//永久解锁动态码
IF(receive_data101[1]=16#21)THEN
	swGpsPrivate.caculateCodeH(code1:=CANO_engine_hour_h,code2:=TO_DINT(CANO_engine_hour_m),result =>CANO_DONGTAIMA1);
	swGpsPrivate.caculateCodeL(code1:=x1,code2:=x2,result =>CANO_DONGTAIMA2);
	send_data102[0]:=receive_data101[0];
	send_data102[1]:=16#21;
	send_data102[2]:=DINT_TO_BYTE((CANO_DONGTAIMA1 MOD 65536) MOD 256);
	send_data102[3]:=DINT_TO_BYTE((CANO_DONGTAIMA1 MOD 65536)/256);
	send_data102[4]:=DINT_TO_BYTE((CANO_DONGTAIMA1 / 65536) MOD 256);
	send_data102[5]:=DINT_TO_BYTE((CANO_DONGTAIMA2 MOD 65536) MOD 256);
	send_data102[6]:=DINT_TO_BYTE((CANO_DONGTAIMA2 MOD 65536)/256);
	send_data102[7]:=DINT_TO_BYTE((CANO_DONGTAIMA2 / 65536) MOD 256);
	IF tCounter<500 THEN
		tCounter:=tCounter+1;
		CAN1_SEND_102(xEnable:= TRUE, eChannel:= 0, udiID:= 16#102, xExtended:=FALSE, usiDLC:=8 , aData:=send_data102);
	ELSE
		receive_data101[1]:=0;
	END_IF
END_IF
IF(receive_data101[1]=0)THEN
	tCounter:=0;
END_IF
swGpsPrivate.swGpsPermanentCancel(PH:=CANO_DONGTAIMA1,PL:=CANO_DONGTAIMA2,result=>VarGpsYongJiuUnlockPassword2);

END_PROGRAM

// StandardPLC/Application/CAN/CAN1
PROGRAM CAN1
VAR
	CAN2_INTI: ifmRCAN.CAN_Enable;
	CANO_FUEL1 :UINT;
	CANO_FUEL2 :UINT;
	Idling_OK_biaozhi:BOOL;
	TIME_20ms:TON;
	TIME_30ms:ton;
	TIME_500ms:ton;
	TIME_5000ms:TON;
	TIME_3000ms:TON;
	TIME_1000ms:TON;
	TIME_BUTTON1:TON;
	TIME_BUTTON2:TON;
	TIME_BIAOZHI1:TON;
	TIME_GPSCAN_ERROR:TON;
	CAN2_RECE_1:ifmRCAN.CAN_Rx;
	CAN2_RECE_2:ifmRCAN.CAN_Rx;
	CAN2_RECE_3:ifmRCAN.CAN_Rx;
	CAN2_RECE_4:ifmRCAN.CAN_Rx;
	CAN2_RECE_5:ifmRCAN.CAN_Rx;
	CAN2_RECE_6:ifmRCAN.CAN_Rx;
	CAN2_RECE_7:ifmRCAN.CAN_Rx;
	CAN2_RECE_8:ifmRCAN.CAN_Rx;
	CAN2_RECE_9:ifmRCAN.CAN_Rx;
	CAN2_rece_data18FD7C00:ifmRCAN.CAN_Rx;
	CAN2_rece_data18FEFF00:ifmRCAN.CAN_Rx;
	CAN2_rece_data18FE5600:ifmRCAN.CAN_Rx;
	CAN2_SEND_000:ifmRCAN.CAN_Tx;
	CAN2_SEND_300:ifmRCAN.CAN_Tx;
	CAN2_SEND_1:ifmRCAN.CAN_Tx;
	CAN2_SEND_2:ifmRCAN.CAN_Tx;
	CAN2_SEND_3:ifmRCAN.CAN_Tx;
	CAN2_SEND_4:ifmRCAN.CAN_Tx;
	CAN2_SEND_5:ifmRCAN.CAN_Tx;
	CAN2_SEND_6:ifmRCAN.CAN_Tx;
	CAN2_SEND_7:ifmRCAN.CAN_Tx;
	CAN2_SEND_8:ifmRCAN.CAN_Tx;
	CAN2_SEND_9:ifmRCAN.CAN_Tx;
	CAN2_SEND_10:ifmRCAN.CAN_Tx;


	rece_data18FEEF00: ARRAY [0..7] OF USINT;
	rece_data0CF00400: ARRAY [0..7] OF USINT;
	rece_data18FEE500: ARRAY [0..7] OF USINT;
	rece_data18FEE900: ARRAY [0..7] OF USINT;
	rece_data0CF00300: ARRAY [0..7] OF USINT;
	rece_data18FEEE00: ARRAY [0..7] OF USINT;
	rece_data18FEF200: ARRAY [0..7] OF USINT;
	
	rece_data18FD7C00: ARRAY [0..7] OF USINT;
	rece_data18FEFF00: ARRAY [0..7] OF USINT;
	rece_data18FE5600: ARRAY [0..7] OF USINT;

	rece_data5: ARRAY [0..7] OF USINT;
	rece_data7: ARRAY [0..7] OF USINT;
	rece_data8: ARRAY [0..7] OF USINT;
	send_data000:ARRAY [0..7] OF USINT;
	send_data1:ARRAY [0..7] OF USINT;
	send_data2:ARRAY [0..7] OF USINT;
	send_data3:ARRAY [0..7] OF USINT;
	send_data4:ARRAY [0..7] OF USINT;
	send_data5:ARRAY [0..7] OF USINT;
	
	send_data300:ARRAY [0..7] OF USINT;	
	send_data300_1:ARRAY [0..7] OF USINT;
	Byte1_1: BYTE;
	Byte2_1: BYTE;
	Byte3_1: BYTE;
	Byte4_1: BYTE;
	Byte5_1: BYTE;
	Byte1_2: BYTE;
	Byte2_2: BYTE;
	Byte3_2: BYTE;
	Byte4_2: BYTE;
	Byte1_3: BYTE;
	Byte2_3: BYTE;
	Byte3_3: BYTE;
	Byte4_3: BYTE;
	Byte1_4: BYTE;
	Byte2_4: BYTE;
	Byte3_4: BYTE;
	Byte4_4: BYTE;
	Byte1_5: BYTE;
	Byte2_5: BYTE;
	Byte3_5: BYTE;
	Byte4_5: BYTE;
	Byte1_6: BYTE;
	Byte2_6: BYTE;
	Byte3_6: BYTE;
	Byte4_6: BYTE;
	Byte1_7: BYTE;
	Byte2_7: BYTE;
	Byte3_7: BYTE;
	Byte4_7: BYTE;
	Byte1_8: BYTE;
	Byte2_8: BYTE;
	Byte3_8: BYTE;
	Byte4_8: BYTE;
	Byte1_9: BYTE;
	Byte2_9: BYTE;
	Byte3_9: BYTE;
	Byte4_9: BYTE;
	Byte1_10: BYTE;
	Byte2_10: BYTE;
	Byte3_10: BYTE;
	Byte4_10: BYTE;
	Byte_x1:BYTE;
	Byte_x2:BYTE;
	byte_x3:BYTE;
	Byte_x4:BYTE;
	byte_x5:BYTE;
	Byte_x6:BYTE;
	byte_x7:BYTE;
	Codes_N:BYTE;
	
    Counter1:BYTE;
    Counter2:BYTE;
    Counter3:BYTE;
(*******GPS**********)
	NewGpsRealFakeTargetData: UINT;
	CAN2_RECE_GPS200:ifmRCAN.CAN_Rx;
	receive_data200:ARRAY [0..7] OF USINT;
	
	F1: F_TRIG;
	F2: F_TRIG;
	F3: F_TRIG;
	F4: F_TRIG;
	TIME_600S:TON;
	TIME_300S:TON;
	TIME_1S:TON;
	TT3:TON;
	CANO_water_tem_1:UINT;
	GPS_CAN_ERROR_1: BOOL;
	archives:UINT;
	
	CANO_X_OFFSET: UINT;
	CANO_Y_OFFSET: UINT;
	MastWorkMode: BOOL;
	GPSYONGJIU:TMP.Passward;
	GPSYOONGJIUJIESUO:DINT;
	Input_minute: INT;
	Xangle:REAL;
	Yangle:REAL;
	X_Offset_zhongjian: REAL;
	Y_Offset_zhongjian: REAL;
	Y_Offset: UINT;
	X_Offset: UINT;
	PWM_Y34_SET_Target: INT;
	CANO_DonglitouPressure_last: INT;
	send_data6: ARRAY [0..7] OF USINT;
	send_data7: ARRAY [0..7] OF USINT;
	send_data8: ARRAY [0..7] OF USINT;
	send_data9: ARRAY [0..7] OF USINT;
	send_data10: ARRAY [0..7] OF USINT;
	
	AI_ECM2_9_last:UINT;
	speed_enable_jinzhi:BOOL;
	EngineSpeedTarget_last:UINT;
	stop_value:BYTE;
	over_value:BYTE;
	
	ZAISHENG_LIGHT1: BYTE;
	ZAISHENG_LIGHT2: BYTE;
	VarZaiSheng_light_A:BOOL;
	VarZaiSheng_light_B:BOOL;
	ZAISHENG_LIGHT3: BYTE;
	ZAISHENG_LIGHT4: BYTE;

	JINZHI_LIGHT1: BYTE;
	DEF_LIGHT1: BYTE;
	DEF_LIGHT2: BYTE;
	GAOPAIWEN_LIGHT1: BYTE;
	BL:BLINK;
	sCounter:BYTE;
	fcounter:byte;
	
END_VAR

(*CAN2口使能及初始化*)
CAN2_INTI(xEnable:=NOT init_1 , eChannel:=ifmRCAN.ifmDevice.CHAN_1, eBaudrate:=ifmRCAN.ifmDevice.CAN_BAUDRATE.KBAUD_250 );	

(*CAN2口 接倾角传感器 发动机 GPS *)
send_data000[0]:=16#01;
send_data000[1]:=16#00;
CAN2_SEND_000(xEnable:= TIME_5000ms.Q, eChannel:= 1, udiID:= 16#000, xExtended:=FALSE, usiDLC:=2 , aData:=send_data000 );

(****************发动机接收/发动数据*******************)
//发动机水温(*FROM 18FEEE00*)
CAN2_RECE_1(xEnable:=TRUE , eChannel:= 1, xExtended:= TRUE, aData=> rece_data18FEEE00, udiID:= 16#18FEEE00);
CANO_water_tem:=(rece_data18FEEE00[0])-40;
IF CANO_water_tem<=0 THEN
	CANO_water_tem:=0;
END_IF
CANO_water_tem_1:=INT_TO_UINT(CANO_water_tem);
IF (CANO_water_tem_1 > PAR_WarnWaterTem_High) THEN
	CANO_TooHigh_WaterTem:=TRUE;
ELSE
	CANO_TooHigh_WaterTem:=FALSE;
END_IF
//机油压力
CAN2_RECE_2(xEnable:=TRUE , eChannel:= 1, xExtended:= TRUE, aData=> rece_data18FEEF00, udiID:= 16#18FEEF00);
CANO_Lub_Press:=REAL_TO_UINT(USINT_TO_REAL(rece_data18FEEF00[3])*2/5);

IF(CANO_Lub_Press<PAR_WarnOilPress_Low AND CANO_SPEED>500)THEN
	CANO_TooLow_OilPress :=TRUE;
ELSE
	CANO_TooLow_OilPress :=FALSE;
END_IF

//发动机转速(*FROM 0CF00400  *)
CAN2_RECE_3(xEnable:=TRUE , eChannel:= 1, xExtended:= TRUE, aData=> rece_data0CF00400, udiID:= 16#0CF00400);
CANO_SPEED:=REAL_TO_UINT((rece_data0CF00400[4]*256+rece_data0CF00400[3])/8);

//发动机负荷率
CAN2_RECE_4(xEnable:=TRUE , eChannel:= 1, xExtended:= TRUE, aData=> rece_data0CF00300, udiID:= 16#0CF00300);
CANO_LoadRate:=rece_data0CF00300[2];

//发送机燃油消耗
CAN2_RECE_6(xEnable:=TRUE , eChannel:= 1, xExtended:= TRUE, aData=> rece_data18FEE900, udiID:= 16#18FEE900);
CANO_FUEL1:=REAL_TO_UINT((BYTE_TO_REAL(rece_data18FEE900[0])+BYTE_TO_REAL(rece_data18FEE900[1])*256));
CANO_FUEL2:=REAL_TO_UINT((BYTE_TO_REAL(rece_data18FEE900[2])+BYTE_TO_REAL(rece_data18FEE900[3])*256));
CANO_Accumu_Fuel_2:=REAL_TO_UDINT((UINT_TO_REAL(CANO_FUEL1)+65536*UINT_TO_REAL(CANO_FUEL2))*0.5);
(*累计油耗清零*)
IF(CANI_Button_RecordClear AND CANO_Accumu_Fuel_2<1000) THEN
	Par_Accumu_Fuel_1:=CANO_Accumu_Fuel_2;
END_IF

IF(CANO_Accumu_Fuel_2>=Par_Accumu_Fuel_1) THEN
	CANO_Accumu_Fuel:=CANO_Accumu_Fuel_2 - Par_Accumu_Fuel_1;
ELSE
	CANO_Accumu_Fuel:=CANO_Accumu_Fuel_2;
END_IF

//发动机瞬间油耗
CAN2_RECE_9(xEnable:=TRUE , eChannel:= 1, xExtended:= TRUE, aData=> rece_data18FEF200, udiID:= 16#18FEF200);
FuelMomentary1 := rece_data18FEF200[1]*256 + rece_data18FEF200[0];
FuelMomentary  := FuelMomentary1/2;

(*发动机故障代码检测*)
CAN2_RECE_5(xEnable:=TRUE , eChannel:= 1, xExtended:= TRUE, aData=> rece_data5, udiID:= 16#18FECA00);(*单故障*)
CAN2_RECE_8(xEnable:=TRUE , eChannel:= 1, xExtended:= TRUE, aData=> rece_data8, udiID:= 16#18ECFF00);(*多故障  火车头*)
CAN2_RECE_7(xEnable:=TRUE , eChannel:= 1, xExtended:= TRUE, aData=> rece_data7, udiID:= 16#18EBFF00);(*多故障  火车车厢*)

(*发动机故障代码解析，包括故障对象SPN（19位）和故障类型FMI（5位）两部分，三个字节*)
(*存在多个故障时*)
IF(rece_data8[5] = 16#CA) AND (rece_data8[6] = 16#FE)  AND  (rece_data8[7] = 16#00) THEN(*表示有多故障*)
	Codes_N :=WORD_TO_BYTE(((rece_data8[1]+rece_data8[2]*256)-2)/4);(*故障个数计算*)
	IF	rece_data7[0] = 16#01  THEN   (*第一个数据包*)
		IF	rece_data7[6] >= 16#80 THEN
			Byte5_1 := rece_data7[7];
			Byte4_1 := SHR(rece_data7[3],5);(*SPN第3个字节*)
			Byte3_1 := SHL(rece_data7[3],3) +SHR(rece_data7[4],5) ;(*SPN第2个字节*)
			Byte2_1 := SHL(rece_data7[4],3) +SHR(rece_data7[5],5) ;(*SPN第1个字节*)
			Byte1_1 := rece_data7[5]  AND 2#00011111 ;(*计算FMI*)
			Codes_SPN[1] := BYTE_TO_UDINT( Byte4_1)*65536 +BYTE_TO_UDINT( Byte3_1)*256 +BYTE_TO_UDINT( Byte2_1);
			Codes_FMI[1] :=  Byte1_1;
		END_IF
		IF	rece_data7[6] < 16#80 THEN
			Byte5_1 := rece_data7[7];
			Byte4_1 := SHR(rece_data7[5],5);
			Byte3_1 := rece_data7[4] ;
			Byte2_1 := rece_data7[3] ;
			Byte1_1 := rece_data7[5]  AND 2#00011111 ;
			Codes_SPN[1] := BYTE_TO_UDINT( Byte4_1)*65536 +BYTE_TO_UDINT( Byte3_1)*256 +BYTE_TO_UDINT( Byte2_1);
			Codes_FMI[1] :=  Byte1_1;
		END_IF
	END_IF
	IF	rece_data7[0] = 16#02  THEN  (*第二个数据包*)
		IF	rece_data7[3] >= 16#80 THEN
			Byte4_2 := SHR(Byte5_1,5);
			Byte3_2 := SHL(Byte5_1,3) +SHR(rece_data7[1],5) ;
			Byte2_2 := SHL(rece_data7[1],3) +SHR(rece_data7[2],5) ;
			Byte1_2 := rece_data7[2]  AND 2#00011111 ;
			IF  rece_data7[4]=16#FF AND rece_data7[5]=16#FF AND rece_data7[6]=16#FF AND rece_data7[7]=16#FF THEN
				Byte4_3:=0;
				Byte3_3:=0;
				Byte2_3:=0;
				Byte1_3:=0;
				Codes_N:=2;
				Codes_SPN[2] := BYTE_TO_UDINT( Byte4_2)*65536 +BYTE_TO_UDINT( Byte3_2)*256 +BYTE_TO_UDINT( Byte2_2);
				Codes_FMI[2]:=  Byte1_2;
			ELSE
				Byte4_3 := SHR(rece_data7[4],5);
				Byte3_3 := SHL(rece_data7[4],3) +SHR(rece_data7[5],5) ;
				Byte2_3 := SHL(rece_data7[5],3) +SHR(rece_data7[6],5) ;
				Byte1_3 := rece_data7[6]  AND 2#00011111 ;
				Codes_N:=3;
				Codes_SPN[3] := BYTE_TO_UDINT( Byte4_3)*65536 +BYTE_TO_UDINT( Byte3_3)*256 +BYTE_TO_UDINT( Byte2_3);
				Codes_FMI[3]:=  Byte1_3;
			END_IF
		END_IF
		IF	rece_data7[3] < 16#80 THEN
			IF  rece_data7[4]=16#FF AND rece_data7[5]=16#FF AND rece_data7[6]=16#FF AND rece_data7[7]=16#FF THEN
				Codes_N:=2;
				Byte4_2 := SHR(rece_data7[2],5);
				Byte3_2 := rece_data7[1] ;
				Byte2_2 := Byte5_1 ;
				Byte1_2 := rece_data7[2]  AND 2#00011111 ;
				Codes_SPN[2] := BYTE_TO_UDINT( Byte4_2)*65536 +BYTE_TO_UDINT( Byte3_2)*256 +BYTE_TO_UDINT( Byte2_2);
				Codes_FMI[2] :=  Byte1_2;
			ELSE
				Codes_N:=3;
				Byte4_3 := SHR(rece_data7[6],5);
				Byte3_3 := rece_data7[5] ;
				Byte2_3 := rece_data7[4] ;
				Byte1_3 := rece_data7[6]  AND 2#00011111 ;
				Codes_SPN[3] := BYTE_TO_UDINT( Byte4_3)*65536 +BYTE_TO_UDINT( Byte3_3)*256 +BYTE_TO_UDINT( Byte2_3);
				Codes_FMI[3] :=  Byte1_3;
			END_IF
		END_IF
	END_IF
	IF	rece_data7[0] = 16#03  THEN  (*第三个数据包*)
		IF	rece_data7[4] >= 16#80 THEN
			Byte4_4 := SHR(rece_data7[1],5);
			Byte3_4 := SHL(rece_data7[1],3) +SHR(rece_data7[2],5) ;
			Byte2_4 := SHL(rece_data7[2],3) +SHR(rece_data7[3],5) ;
			Byte1_4 := rece_data7[3]  AND 2#00011111 ;
		ELSIF rece_data7[4] < 16#80 THEN
			Byte4_4 := SHR(rece_data7[3],5);
			Byte3_4 := rece_data7[2] ;
			Byte2_4 := rece_data7[1] ;
			Byte1_4 := rece_data7[3]  AND 2#00011111 ;
		END_IF
			Codes_SPN[4] := BYTE_TO_UDINT( Byte4_4)*65536 +BYTE_TO_UDINT( Byte3_4)*256 +BYTE_TO_UDINT( Byte2_4);
			Codes_FMI[4] :=  Byte1_4;
		IF  rece_data7[5]=16#FF AND rece_data7[6]=16#FF AND rece_data7[7]=16#FF  THEN
				Byte4_5:=0;
				Byte3_5:=0;
				Byte2_5:=0;
				Byte1_5:=0;
				Codes_N:=4;
		ELSE
				Codes_N:=5;
				IF	Byte_x1 >= 16#80 THEN
					Byte4_5 := SHR(rece_data7[5],5);
					Byte3_5 := SHL(rece_data7[5],3) +SHR(rece_data7[6],5) ;
					Byte2_5 := SHL(rece_data7[6],3) +SHR(rece_data7[7],5) ;
					Byte1_5 := rece_data7[7]  AND 2#00011111 ;
				ELSIF Byte_x1 < 16#80 THEN
					Byte4_5 := SHR(rece_data7[7],5);
					Byte3_5 := rece_data7[6] ;
					Byte2_5 := rece_data7[5] ;
					Byte1_5 := rece_data7[7]  AND 2#00011111 ;
				END_IF
					Codes_SPN[5] := BYTE_TO_UDINT( Byte4_5)*65536 +BYTE_TO_UDINT( Byte3_5)*256 +BYTE_TO_UDINT( Byte2_5);
					Codes_FMI[5] :=  Byte1_5;
		END_IF
	END_IF
	IF	rece_data7[0] = 16#04  THEN  (*第4个数据包*)
			Byte_x1:=rece_data7[1];
		IF	rece_data7[5] >= 16#80 THEN
			Byte4_6 := SHR(rece_data7[2],5);
			Byte3_6 := SHL(rece_data7[2],3) +SHR(rece_data7[3],5) ;
			Byte2_6 := SHL(rece_data7[3],3) +SHR(rece_data7[4],5) ;
			Byte1_6 := rece_data7[4]  AND 2#00011111 ;
		ELSIF rece_data7[4] < 16#80 THEN
			Byte4_6 := SHR(rece_data7[4],5);
			Byte3_6 := rece_data7[3] ;
			Byte2_6 := rece_data7[2] ;
			Byte1_6 := rece_data7[4]  AND 2#00011111 ;
		END_IF
			Codes_SPN[6] := BYTE_TO_UDINT( Byte4_6)*65536 +BYTE_TO_UDINT( Byte3_6)*256 +BYTE_TO_UDINT( Byte2_6);
			Codes_FMI[6] :=  Byte1_6;
		IF  rece_data7[6]=16#FF AND rece_data7[7]=16#FF  THEN
				Byte4_7:=0;
				Byte3_7:=0;
				Byte2_7:=0;
				Byte1_7:=0;
				Codes_N:=6;
		ELSE
				Codes_N:=7;
				IF	Byte_x2 >= 16#80 THEN
					Byte4_7 := SHR(rece_data7[6],5);
					Byte3_7 := SHL(rece_data7[6],3) +SHR(rece_data7[7],5) ;
					Byte2_7 := SHL(rece_data7[7],3) +SHR(Byte_x3,5) ;
					Byte1_7 := Byte_x3  AND 2#00011111 ;
				ELSIF Byte_x2 < 16#80 THEN
					Byte4_7 := SHR(Byte_x3,5);
					Byte3_7 := rece_data7[7] ;
					Byte2_7 := rece_data7[6] ;
					Byte1_7 := Byte_x3  AND 2#00011111 ;
				END_IF
					Codes_SPN[7] := BYTE_TO_UDINT( Byte4_7)*65536 +BYTE_TO_UDINT( Byte3_7)*256 +BYTE_TO_UDINT( Byte2_7);
					Codes_FMI[7] :=  Byte1_7;
		END_IF
	END_IF
	IF	rece_data7[0] = 16#05  THEN  (*第5个数据包*)
			Byte_x2:=rece_data7[2];
			Byte_x3:=rece_data7[1];
		IF	rece_data7[6] >= 16#80 THEN
			Byte4_8 := SHR(rece_data7[3],5);
			Byte3_8 := SHL(rece_data7[3],3) +SHR(rece_data7[4],5) ;
			Byte2_8 := SHL(rece_data7[4],3) +SHR(rece_data7[5],5) ;
			Byte1_8 := rece_data7[5]  AND 2#00011111 ;
		ELSIF rece_data7[6] < 16#80 THEN
			Byte4_8 := SHR(rece_data7[5],5);
			Byte3_8 := rece_data7[4] ;
			Byte2_8 := rece_data7[3] ;
			Byte1_8 := rece_data7[5]  AND 2#00011111 ;
		END_IF
			Codes_SPN[8] := BYTE_TO_UDINT( Byte4_8)*65536 +BYTE_TO_UDINT( Byte3_8)*256 +BYTE_TO_UDINT( Byte2_8);
			Codes_FMI[8] :=  Byte1_8;
		IF  rece_data7[7]=16#FF  THEN
				Byte4_9:=0;
				Byte3_9:=0;
				Byte2_9:=0;
				Byte1_9:=0;
				Codes_N:=8;
		ELSE
				Codes_N:=9;
				IF	Byte_x4 >= 16#80 THEN
					Byte4_9 := SHR(rece_data7[7],5);
					Byte3_9 := SHL(rece_data7[7],3) +SHR(Byte_x5,5) ;
					Byte2_9 := SHL(Byte_x5,3) +SHR(Byte_x6,5) ;
					Byte1_9 := Byte_x6  AND 2#00011111 ;
				ELSIF Byte_x4 < 16#80 THEN
					Byte4_9 := SHR(Byte_x6,5);
					Byte3_9 := Byte_x5 ;
					Byte2_9 := rece_data7[7] ;
					Byte1_9 := Byte_x6  AND 2#00011111 ;
				END_IF
					Codes_SPN[9] := BYTE_TO_UINT( Byte4_9)*65536 +BYTE_TO_UINT( Byte3_9)*256 +BYTE_TO_UINT( Byte2_9);
					Codes_FMI[9] :=  Byte1_9;
		END_IF
	END_IF
	IF	rece_data7[0] = 16#06  THEN  (*第6个数据包*)
			Codes_N:=10;
			Byte_x4:=rece_data7[3];
			Byte_x5:=rece_data7[1];
			Byte_x6:=rece_data7[2];
		IF	rece_data7[7] >= 16#80 THEN
			Byte4_10 := SHR(rece_data7[4],5);
			Byte3_10 := SHL(rece_data7[4],3) +SHR(rece_data7[5],5) ;
			Byte2_10 := SHL(rece_data7[5],3) +SHR(rece_data7[6],5) ;
			Byte1_10 := rece_data7[6]  AND 2#00011111 ;
		ELSIF rece_data7[6] < 16#80 THEN
			Byte4_10 := SHR(rece_data7[6],5);
			Byte3_10 := rece_data7[5] ;
			Byte2_10 := rece_data7[4] ;
			Byte1_10 := rece_data7[6]  AND 2#00011111 ;
		END_IF
			Codes_SPN[10] := BYTE_TO_UDINT( Byte4_10)*65536 +BYTE_TO_UDINT( Byte3_10)*256 +BYTE_TO_UDINT( Byte2_10);
			Codes_FMI[10] :=  Byte1_10;
	END_IF
(*只有一个故障时*)
ELSIF rece_data5[5]<>0    THEN
		Codes_N:=1;
		IF	rece_data5[5] >= 16#80 THEN(*1*)
			Byte4_1 := SHR(rece_data5[2],5);
			Byte3_1 := SHL(rece_data5[2],3) +SHR(rece_data5[3],5) ;
			Byte2_1 := SHL(rece_data5[3],3) +SHR(rece_data5[4],5) ;
			Byte1_1 := rece_data5[4]  AND 2#00011111 ;
			Codes_SPN[1] := BYTE_TO_UDINT( Byte4_1)*65536 +BYTE_TO_UDINT( Byte3_1)*256 +BYTE_TO_UDINT( Byte2_1);
			Codes_FMI[1] :=  Byte1_1;
		END_IF
		IF	rece_data5[5] < 16#80 THEN  (*0*)
			Byte4_1 := SHR(rece_data5[4],5);
			Byte3_1 := rece_data5[3] ;
			Byte2_1 := rece_data5[2] ;
			Byte1_1 := rece_data5[4]  AND 2#00011111 ;
			Codes_SPN[1] := BYTE_TO_UDINT( Byte4_1)*65536 +BYTE_TO_UDINT( Byte3_1)*256 +BYTE_TO_UDINT( Byte2_1);
			Codes_FMI[1] :=  Byte1_1;
		END_IF
(*没有故障时*)
ELSE
	Codes_N:=0;
    Codes_SPN[1]:=0;
    Codes_FMI[1]:=0;
END_IF
Codes_SPN_1:=Codes_SPN[1];
Codes_SPN_2:=Codes_SPN[2];
Codes_SPN_3:=Codes_SPN[3];
Codes_SPN_4:=Codes_SPN[4];
Codes_SPN_5:=Codes_SPN[5];
Codes_SPN_6:=Codes_SPN[6];
Codes_SPN_7:=Codes_SPN[7];
Codes_SPN_8:=Codes_SPN[8];
Codes_SPN_9:=Codes_SPN[9];
Codes_SPN_10:=Codes_SPN[10];
Codes_FMI_1:=Codes_FMI[1];
Codes_FMI_2:=Codes_FMI[2];
Codes_FMI_3:=Codes_FMI[3];
Codes_FMI_4:=Codes_FMI[4];
Codes_FMI_5:=Codes_FMI[5];
Codes_FMI_6:=Codes_FMI[6];
Codes_FMI_7:=Codes_FMI[7];
Codes_FMI_8:=Codes_FMI[8];
Codes_FMI_9:=Codes_FMI[9];
Codes_FMI_10:=Codes_FMI[10];
IF(Codes_SPN[1]>9999)THEN Codes_SPN_1:=0;Codes_FMI_1:=0;END_IF
IF(Codes_SPN[2]>9999)THEN Codes_SPN_2:=0;Codes_FMI_2:=0;END_IF
IF(Codes_SPN[3]>9999)THEN Codes_SPN_3:=0;Codes_FMI_3:=0;END_IF
IF(Codes_SPN[4]>9999)THEN Codes_SPN_4:=0;Codes_FMI_4:=0;END_IF
IF(Codes_SPN[5]>9999)THEN Codes_SPN_5:=0;Codes_FMI_5:=0;END_IF
IF(Codes_SPN[6]>9999)THEN Codes_SPN_6:=0;Codes_FMI_6:=0;END_IF
IF(Codes_SPN[7]>9999)THEN Codes_SPN_7:=0;Codes_FMI_7:=0;END_IF
IF(Codes_SPN[8]>9999)THEN Codes_SPN_8:=0;Codes_FMI_8:=0;END_IF
IF(Codes_SPN[9]>9999)THEN Codes_SPN_9:=0;Codes_FMI_9:=0;END_IF
IF(Codes_SPN[10]>9999)THEN Codes_SPN_10:=0;Codes_FMI_10:=0;END_IF

IF Codes_SPN_1=729 AND Codes_FMI_1=3 THEN
	Codes_SPN_1:=0;
	Codes_FMI_1:=0;
END_IF


(*CAN2发送*)
//请求燃油消耗量
TIME_1000ms(IN:=NOT TIME_1000ms.Q,PT:=T#1000MS);
TIME_5000ms(IN:=NOT TIME_5000ms.Q,PT:=T#5000MS);
send_data2[0]:=229;
send_data2[1]:=254;
send_data2[2]:=0;
send_data3[0]:=233;
send_data3[1]:=254;
send_data3[2]:=0;
IF TIME_5000ms.Q THEN
	CAN2_SEND_2(xEnable:= TRUE, eChannel:= 1, udiID:= 16#18EA00F1, xExtended:=TRUE, usiDLC:=8 , aData:=send_data2 );
	CAN2_SEND_3(xEnable:= TRUE, eChannel:= 1, udiID:= 16#18EA00F2, xExtended:=TRUE, usiDLC:=8 , aData:=send_data3 );
END_IF
//发动机转速控制
TIME_BUTTON1(IN:=CANI_Button_YouMen_Min,PT:=T#2S);
TIME_BUTTON2(IN:=CANI_Button_YouMen_Max,PT:=T#2S);
IF(TIME_BUTTON1.Q)THEN
	PAR_YouMen_NegFull:=AI_ECM2_9;
END_IF
IF(TIME_BUTTON2.Q)THEN
	PAR_YouMen_PosFull:=AI_ECM2_9;	
END_IF

IF(PAR_YouMen_PosFull<=PAR_YouMen_NegFull)THEN
	PAR_YouMen_NegFull:=920;
	PAR_YouMen_PosFull:=3200;
END_IF

IF(AI_ECM2_9<PAR_YouMen_NegFull) THEN
	AI_ECM2_9:=PAR_YouMen_NegFull;
END_IF
IF(AI_ECM2_9>PAR_YouMen_PosFull) THEN
	AI_ECM2_9:=PAR_YouMen_PosFull;
END_IF
	//计算油门百分比 	油门分档位
IF(AI_ECM2_9<=1150)THEN
	EngineSpeedTarget := PAR_SpeedLow_Idling;
	AI_ECM2_Flag:=1;
ELSIF(AI_ECM2_9>1150 AND AI_ECM2_9<=1550) THEN
	EngineSpeedTarget := 1200;	
	AI_ECM2_Flag:=2;	
ELSIF(AI_ECM2_9>1550 AND AI_ECM2_9<=2050) THEN
	EngineSpeedTarget := 1450;	
	AI_ECM2_Flag:=3;		
ELSIF(AI_ECM2_9>=2050 AND AI_ECM2_9<=2500) THEN
	EngineSpeedTarget := 1600;
	AI_ECM2_Flag:=4;			
ELSIF(AI_ECM2_9>=2500 AND AI_ECM2_9<=2900) THEN
	EngineSpeedTarget := 1800;
	AI_ECM2_Flag:=5;			
ELSIF(AI_ECM2_9>2900) THEN
	EngineSpeedTarget := PAR_SpeedHigh_Idling;
	AI_ECM2_Flag:=6;			
END_IF

//主卷扬下放时，自动调整转速
IF(PWM_JOYY_L_UP>10 AND AI_ECM2_9>2050 AND (GVL_SaveEngine.SaveEngineMode=1 OR GVL_SaveEngine.SaveEngineMode=8 OR GVL_SaveEngine.SaveEngineMode=11) )THEN
	EngineSpeedTarget:=1500;
END_IF	
//中速开关设定转速
IF(CANI_MidSpeedSwitch)THEN
	IF (PWM_JOYY_L_UP>10) AND (GVL_SaveEngine.SaveEngineMode=1 OR GVL_SaveEngine.SaveEngineMode=8 OR GVL_SaveEngine.SaveEngineMode=11) THEN
		EngineSpeedTarget:=1500;
		AI_ECM2_Flag:=4;
	ELSE
		EngineSpeedTarget:=1600;
	END_IF
END_IF

//模式开关转速设定
(*IF(CANI_MoShiSwitch)THEN
	EngineSpeedTarget:=2100;	
END_IF*)

//自动怠速
IF(CANO_JiayaPressure<60 AND CANO_DonglitouPressure<80 AND CANO_ZhuJuanPressure<60
	AND CANO_MainPUMP_Press1<80 AND CANO_MainPUMP_Press2<80 AND CANO_Fubeng_Press<60) THEN
	Idling_OK_biaozhi:=TRUE;
ELSE
	Idling_OK_biaozhi:=FALSE;		
END_IF
TIME_BIAOZHI1(IN:=Idling_OK_biaozhi,PT:=T#3S);
IF(TIME_BIAOZHI1.Q AND CANI_IdleEnbleSwitch) THEN
	EngineSpeedTarget:=1000;		
END_IF

//GPS Locked

IF(VarGpsSystemLockedState) THEN
	EngineSpeedTarget:=1000;
END_IF

TIME_20ms(IN:=TIME_20ms.Q,PT:=T#10MS);
send_data1[0]:=9;
send_data1[1]:=UINT_TO_BYTE((EngineSpeedTarget*8) MOD 256);
send_data1[2]:=UINT_TO_BYTE((EngineSpeedTarget*8) /256);
send_data1[3]:=0;
send_data1[4]:=255;
send_data1[5]:=255;
send_data1[6]:=255;
send_data1[7]:=255;
//再生灯亮   再生开关打开
	IF((VarHouchuliSwitch=4) AND (ZAISHENG_LIGHT3=1 OR ZAISHENG_LIGHT4=1) AND (EngineSpeedTarget_last=EngineSpeedTarget))THEN
		speed_enable_jinzhi:=TRUE;
	END_IF
	IF(EngineSpeedTarget_last<>EngineSpeedTarget)THEN
		speed_enable_jinzhi:=FALSE;
	END_IF
	IF( NOT  speed_enable_jinzhi)THEN
		CAN2_SEND_1(xEnable:= TRUE, eChannel:= 1, udiID:= 16#0C000003, xExtended:=TRUE, usiDLC:=8 , aData:=send_data1 );
	END_IF		
EngineSpeedTarget_last:=EngineSpeedTarget;
AI_ECM2_9_last:=AI_ECM2_9;

send_data4[0]:=16#E9;
send_data4[1]:=16#FE;
send_data4[2]:=0;
send_data4[3]:=0;
send_data4[4]:=0;
send_data4[5]:=0;
send_data4[6]:=0;
send_data4[7]:=0;
CAN2_SEND_4(xEnable:= TIME_1000ms.Q, eChannel:= 1, udiID:= 16#18EA00F2, xExtended:=TRUE, usiDLC:=8 , aData:=send_data4 );

send_data5[0]:=16#E5;
send_data5[1]:=16#FE;
send_data5[2]:=0;
send_data5[3]:=0;
send_data5[4]:=0;
send_data5[5]:=0;
send_data5[6]:=0;
send_data5[7]:=0;
CAN2_SEND_5(xEnable:= TIME_1000ms.Q, eChannel:= 1, udiID:= 16#18EA00F1, xExtended:=TRUE, usiDLC:=8 , aData:=send_data5 );


send_data7[0]:=16#FF;
send_data7[1]:=16#FF;
send_data7[2]:=16#FF;
send_data7[3]:=16#FF;
send_data7[4]:=16#FF;
send_data7[5]:=VarHouchuliSwitch;
send_data7[6]:=16#FF;
send_data7[7]:=16#FF;

send_data8[0]:=16#FF;
send_data8[1]:=16#FF;
send_data8[2]:=16#FF;
send_data8[3]:=stop_value;
send_data8[4]:=16#FF;
send_data8[5]:=16#FF;
send_data8[6]:=16#FF;
send_data8[7]:=16#FF;

send_data9[0]:=16#FF;
send_data9[1]:=16#FF;
send_data9[2]:=16#00;
send_data9[3]:=16#FF;
send_data9[4]:=16#FF;
send_data9[5]:=16#FF;
send_data9[6]:=16#FF;
send_data9[7]:=16#FF;

TIME_30ms(IN:=NOT TIME_30ms.Q,PT:=T#20MS);
TIME_500ms(IN:=NOT TIME_500ms.Q,PT:=T#500MS);
//发动机停机功能   0CF00130 BYTE3 0---不启用   16#10-停机  间隔30MS
IF (TIME_30ms.Q) THEN
	CAN2_SEND_8(xEnable:= TRUE, eChannel:= 1, udiID:= 16#0CF00130, xExtended:=TRUE, usiDLC:=8 , aData:=send_data8 );
	//SW.fCanSend(SW.eCanChannelType.ch1, 16#0CF00130, SW.eCanIdeType.ext, SW.eCanRtrType.rtrData, send_data8, SendLen);
END_IF
//发动机超越开关  0C850030 BYTE3 0---不启用   1-超越  间隔500MS

IF (TIME_500ms.Q) THEN
	CAN2_SEND_9(xEnable:= TRUE, eChannel:= 1, udiID:= 16#0C850030, xExtended:=TRUE, usiDLC:=8 , aData:=send_data9 ); 
	//SW.fCanSend(SW.eCanChannelType.ch1, 16#0C850030, SW.eCanIdeType.ext, SW.eCanRtrType.rtrData, send_data9, SendLen);
END_IF
IF (TIME_1000ms.Q) THEN
	CAN2_SEND_7(xEnable:= TRUE, eChannel:= 1, udiID:= 16#0CE00030, xExtended:=TRUE, usiDLC:=8 , aData:=send_data7 );
END_IF

//GPS 数据发送
IF(VarMastWorkMode=3)THEN
	MastWorkMode:=TRUE;
ELSE
	MastWorkMode:=FALSE;
END_IF


(*计算x偏移量*)
IF(CANO_ANGLE_X>=9000) THEN
	Xangle:=UINT_TO_REAL(CANO_ANGLE_X - 9000) / 100;
	X_Offset:=REAL_TO_UINT(X_Offset_zhongjian) + 1000;
ELSE
	Xangle:=UINT_TO_REAL(9000 - CANO_ANGLE_X ) / 100;
	X_Offset:=1000 - REAL_TO_UINT(X_Offset_zhongjian);	
END_IF


IF(CANO_ANGLE_Y>=9000) THEN
	Yangle:=UINT_TO_REAL(CANO_ANGLE_Y - 9000) / 100;
	Y_Offset:=REAL_TO_UINT(Y_Offset_zhongjian) + 1000;
ELSE
	Yangle:=UINT_TO_REAL(9000 - CANO_ANGLE_Y ) / 100;
	Y_Offset:=1000 - REAL_TO_UINT(Y_Offset_zhongjian);		
END_IF

IF(CANO_DEPTH>1000)THEN
	X_Offset_zhongjian:= TAN(Xangle*3.14/180) * (UINT_TO_REAL(CANO_DEPTH ) - 1000);
	Y_Offset_zhongjian:= TAN(Yangle*3.14/180) * (UINT_TO_REAL(CANO_DEPTH ) - 1000);
ELSE
	X_Offset_zhongjian:=0;
	Y_Offset_zhongjian:=0;
END_IF
IF X_Offset_zhongjian>50 THEN
	X_Offset_zhongjian:=50;
END_IF
IF Y_Offset_zhongjian>50 THEN
	Y_Offset_zhongjian:=50;
END_IF

IF(CANO_DonglitouPressure>280) THEN
	CANO_PowerSpeed :=250;
	CANO_PowerNiuJu :=8;
ELSIF(CANO_DonglitouPressure>270) THEN   
	CANO_PowerSpeed :=225;
	CANO_PowerNiuJu :=8;
ELSIF(CANO_DonglitouPressure>260) THEN   
	CANO_PowerSpeed :=198;
	CANO_PowerNiuJu :=9;
ELSIF(CANO_DonglitouPressure>250) THEN   
	CANO_PowerSpeed :=175;
	CANO_PowerNiuJu :=9;
ELSIF(CANO_DonglitouPressure>240) THEN   
	CANO_PowerSpeed :=153;
	CANO_PowerNiuJu :=10;
ELSIF(CANO_DonglitouPressure>230) THEN   
	CANO_PowerSpeed :=132;
	CANO_PowerNiuJu :=11;
ELSIF(CANO_DonglitouPressure>220) THEN   
	CANO_PowerSpeed :=112;
	CANO_PowerNiuJu :=12;
ELSIF(CANO_DonglitouPressure>210) THEN   
	CANO_PowerSpeed :=93;
	CANO_PowerNiuJu :=15;
ELSIF(CANO_DonglitouPressure>200) THEN   
	CANO_PowerSpeed :=76;
	CANO_PowerNiuJu :=18;
ELSIF(CANO_DonglitouPressure>190) THEN   
	CANO_PowerSpeed :=59;
	CANO_PowerNiuJu :=22;
ELSIF(CANO_DonglitouPressure<190 AND CANO_DonglitouPressure>=20) THEN
	CANO_PowerSpeed :=CANO_DonglitouPressure * 2 /10;
	CANO_PowerNiuJu :=28;
ELSIF(  CANO_DonglitouPressure<20)THEN
	CANO_PowerSpeed :=0;
	CANO_PowerNiuJu :=0;
END_IF



//国四发动机指示灯

CAN2_rece_data18FD7C00(xEnable:=TRUE , eChannel:= 1, xExtended:= TRUE, aData=> rece_data18FD7C00, udiID:= 16#18FD7C00);
CAN2_rece_data18FEFF00(xEnable:=TRUE , eChannel:= 1, xExtended:= TRUE, aData=> rece_data18FEFF00, udiID:= 16#18FEFF00);
CAN2_rece_data18FE5600(xEnable:=TRUE , eChannel:= 1, xExtended:= TRUE, aData=> rece_data18FE5600, udiID:= 16#18FE5600);

ZAISHENG_LIGHT1:=rece_data18FD7C00[1] AND 2#00000100;  (* //0x04 *)
ZAISHENG_LIGHT2:=rece_data18FD7C00[1] AND 2#00001000;   (*//0x08 *)
IF ZAISHENG_LIGHT1=4 OR ZAISHENG_LIGHT2=8 THEN (*  //a判断 *)
	VarZaiSheng_light_A:=FALSE;
ELSE
	VarZaiSheng_light_A:=TRUE;
END_IF
IF VarZaiSheng_light_A  THEN                 (*  //b判断<<5,左移5位，保留低3位 *)
	VarZaiSheng_light_B:= BYTE_TO_BOOL(rece_data18FD7C00[6] AND 2#00000111);
ELSE
	VarZaiSheng_light_B:=FALSE;
END_IF

BL(ENABLE:=TRUE,TIMELOW:=T#0.5S,TIMEHIGH:=T#0.5S);
IF VarZaiSheng_light_A AND (NOT VarZaiSheng_light_B) THEN
	ZAISHENG_LIGHT:=BL.OUT;   (*//再生灯闪烁(频率1Hz)*)
END_IF

ZAISHENG_LIGHT3:=rece_data18FD7C00[0] AND 2#00000001;    (*//0x01 *)
ZAISHENG_LIGHT4:=rece_data18FD7C00[0] AND 2#00000100;   (* //0x04 *)
IF(NOT VarZaiSheng_light_A) OR VarZaiSheng_light_B THEN
	IF ZAISHENG_LIGHT3=1 THEN
		ZAISHENG_LIGHT:=TRUE;      (*  //再生灯亮*)
	ELSE
		ZAISHENG_LIGHT:=FALSE;       (*//再生灯不亮 *)
	END_IF
	IF ZAISHENG_LIGHT4=4 THEN	
		ZAISHENG_LIGHT:=BL.OUT;    (*//再生灯闪烁(频率1Hz)*)
	END_IF

END_IF

(*再生禁止灯*)
JINZHI_LIGHT1:=(rece_data18FD7C00[2] AND 2#00000100);    (*//0x04 *)
IF JINZHI_LIGHT1=4 THEN
	JINZHI_LIGHT:=TRUE;
ELSE
	JINZHI_LIGHT:=FALSE;
END_IF

(*高排温灯*)
GAOPAIWEN_LIGHT1:=(rece_data18FD7C00[6] AND 2#00000100);   (* //0x04 *)
IF GAOPAIWEN_LIGHT1=4 THEN
	GAOPAIWEN_LIGHT:=TRUE;
ELSE
	GAOPAIWEN_LIGHT:=FALSE;
END_IF


IF rece_data18FE5600[0]  <= 250  THEN
	urea_level:=REAL_TO_BYTE(BYTE_TO_REAL(rece_data18FE5600[0])*0.4);(*尿素液位*)
END_IF
(*def灯*)
DEF_LIGHT1:=(rece_data18FE5600[4] AND 2#00100000);   (*//0x20(*点亮*)*)
DEF_LIGHT2:=(rece_data18FE5600[4] AND 2#10000000);    (*//0x80(*闪烁*)*)
IF DEF_LIGHT1=32 AND  DEF_LIGHT2<>128 THEN
	DEF_LIGHT:=TRUE;         (*DEF灯亮 *)
ELSIF DEF_LIGHT1<>32 AND DEF_LIGHT2=128 THEN
	DEF_LIGHT:=BL.OUT;       (*//DEF灯闪烁	*)
ELSE
	DEF_LIGHT:=FALSE;
END_IF

(*驾驶员警告灯*)
IF BYTE_TO_BOOL(rece_data18FEFF00[1] AND 2#00000001) THEN
	JIASHIYUANWARN_LIGHT:=TRUE;
ELSIF BYTE_TO_BOOL(rece_data18FEFF00[1] AND 2#00000100)THEN
	JIASHIYUANWARN_LIGHT:=BL.OUT;   (*频率1Hz*)
ELSE
	JIASHIYUANWARN_LIGHT:=FALSE;
END_IF




//后处理显示器开关逻辑
IF VarZaishengjinzhiSwitch THEN
	VarHouchuliSwitch:=1;
ELSIF((NOT VarZaishengjinzhiSwitch ) AND VarQiangzhiZaishengSwitch) THEN
	VarHouchuliSwitch:=4;
ELSIF((NOT VarZaishengjinzhiSwitch ) AND (NOT VarQiangzhiZaishengSwitch))THEN
	VarHouchuliSwitch:=0;
END_IF

END_PROGRAM

// StandardPLC/Application/CAN/GPS_TONGXING_ALL
PROGRAM GPS_TONGXING_ALL
VAR
	TIME_100ms:TON;
	TIME_500ms:TON;
	TIME_510ms:TON;
	TIME_520ms:TON;
	TIME_530ms:TON;
	TIME_1000ms:TON;
	TIME_1000ms_2:TON;
	TIME_2s:TON;
	TIME_60S:TON;
	TIME_1S_1:TON;
	TIME_60s_2:TON;
	TIME_10s:TON;
	TIME_5s:TON;
	SendLen : BYTE := 8;
	count:UINT;
	WORK_SEND:BOOL;
	(*控制器状态字*)
	VarCanGpsLockCommand_A1:BOOL;(*锁车指令状态*)
	VarCanGpsLockCommand_B1:BOOL;(*锁车指令状态*)
	VarCanGpsLockCommand_C1:BOOL;(*锁车指令状态*)
	VarCanGpsLockCommand_D1:BOOL;(*锁车指令状态*)
	VarCanGpsLockCommand_E1:BOOL;(*锁车指令状态*)
	send_data200:ARRAY [0..7] OF USINT;
	send_data201:ARRAY [0..7] OF USINT;
	send_data202:ARRAY [0..7] OF USINT;
	send_data203:ARRAY [0..7] OF USINT;
	send_data204:ARRAY [0..7] OF USINT;
	send_data205:ARRAY [0..7] OF USINT;
	send_data206:ARRAY [0..7] OF USINT;
	send_data207:ARRAY [0..7] OF USINT;
	send_data208:ARRAY [0..7] OF USINT;
	send_data209:ARRAY [0..7] OF USINT;
	send_data20A:ARRAY [0..7] OF USINT;
	send_data20B:ARRAY [0..7] OF USINT;
	send_data20C:ARRAY [0..7] OF USINT;
	send_data20D:ARRAY [0..7] OF USINT;
	send_data20E:ARRAY [0..7] OF USINT;
	send_data20F:ARRAY [0..7] OF USINT;
	send_data2FF:ARRAY [0..7] OF USINT;

	send_data210:ARRAY [0..7] OF USINT;
	send_data211:ARRAY [0..7] OF USINT;
	send_data212:ARRAY [0..7] OF USINT;
	send_data213:ARRAY [0..7] OF USINT;
	send_data214:ARRAY [0..7] OF USINT;
	send_data215:ARRAY [0..7] OF USINT;
	send_data216:ARRAY [0..7] OF USINT;
	send_data217:ARRAY [0..7] OF USINT;
	send_data218:ARRAY [0..7] OF USINT;
	send_data219:ARRAY [0..7] OF USINT;
	send_data220:ARRAY [0..7] OF USINT;
	send_data2C0:ARRAY [0..7] OF USINT;
	send_data2E0:ARRAY [0..7] OF USINT;
	send_data2F0:ARRAY [0..7] OF USINT;
(*向远程平台发送数据*)
	send_data280:ARRAY [0..7] OF USINT;
	send_data281:ARRAY [0..7] OF USINT;
	send_data282:ARRAY [0..7] OF USINT;
	send_data283:ARRAY [0..7] OF USINT;
	send_data284:ARRAY [0..7] OF USINT;
	send_data285:ARRAY [0..7] OF USINT;
	send_data2B0:ARRAY [0..7] OF USINT;
	send_data2B1:ARRAY [0..7] OF USINT;
	send_data18FF0001:ARRAY [0..7] OF USINT;
	
(*物联网终端状态字*)
	STATE_WARN:BOOL;
	STATE_Satellite:BOOL;
	STATE_ACC:BOOL;
	STATE_WarnConnection:BOOL;
	STATE_WarnPoweroff:BOOL;
	STATE_WarnPowerlow:BOOL;
	STATE_WarnModuleoff:BOOL;
	STATE_WarnTIANXIANoff:BOOL;
	STATE_WarnPowerProtect:BOOL;
	STATE_WarnKAIGAI:BOOL;
	STATE_WarnBAKA:BOOL;
	STATE_Promoteconnect:BOOL;
	STATE_Promoteconnect_20day:BOOL;
	STATE_MASTERSleep:BOOL;
	STATE_BACKUPSleep:BOOL;

(*应答*)
	SN_321:UINT;
	SN_322:UINT;
	SN_323:UINT;(*接收到的323反馈回的序列号*)
	SN_324:UINT;
	SN_325:UINT;
	
	
	CAN1ReceiveFlag13 : BOOL;
	CAN1ReceiveData13 : ARRAY[0..7]OF BYTE;
	CAN1ReceiveLen13 : BYTE;
	CAN1ReceiveFlag14 : BOOL;
	CAN1ReceiveData14 : ARRAY[0..7]OF BYTE;
	CAN1ReceiveLen14 : BYTE;
	CAN1ReceiveFlag15 : BOOL;
	CAN1ReceiveData15 : ARRAY[0..7]OF BYTE;
	CAN1ReceiveLen15 : BYTE;
	CAN1ReceiveFlag16 : BOOL;
	CAN1ReceiveData16 : ARRAY[0..7]OF BYTE;
	CAN1ReceiveLen16 : BYTE;
	CAN1ReceiveFlag17 : BOOL;
	CAN1ReceiveData17 : ARRAY[0..7]OF BYTE;
	CAN1ReceiveLen17 : BYTE;
	CAN1ReceiveFlag18 : BOOL;
	CAN1ReceiveData18 : ARRAY[0..7]OF BYTE;
	CAN1ReceiveLen18 : BYTE;
	CAN1ReceiveFlag22 : BOOL;
	CAN1ReceiveData22 : ARRAY[0..7]OF BYTE;
	CAN1ReceiveLen22 : BYTE;
	CAN1ReceiveFlag23 : BOOL;
	CAN1ReceiveData23 : ARRAY[0..7]OF BYTE;
	CAN1ReceiveLen23 : BYTE;
	ReceiveFlag : BOOL;
	ReceiveData : ARRAY[0..7]OF BYTE;
	ReceiveLen : BYTE;
	
	receive_data300:ARRAY [0..7] OF USINT;
	receive_data303:ARRAY [0..7] OF USINT;
	receive_data320:ARRAY [0..7] OF USINT;
	receive_data321:ARRAY [0..7] OF USINT;
	receive_data322:ARRAY [0..7] OF USINT;
	receive_data323:ARRAY [0..7] OF USINT;
	receive_data324:ARRAY [0..7] OF USINT;
	receive_data325:ARRAY [0..7] OF USINT;
	CLEAR_2C0_SN: UINT;(*2C0发送出去的序列号*)
	CLEAR_Feedback:BOOL;
	clear_trig:R_TRIG;
	Cal_Clear01:UINT;
	Cal_Clear02:BOOL;
	Cal_Clear03:BOOL;
	clear_trig01:R_TRIG;
	CANI_Button_Record_Result_TRIG:BOOL;
	SN_323_Feedback2C0:UINT;
	Result_TRIG:UINT;
	GPSYONGJIU:TMP.Passward;
	GPS_CAN_ERROR_1:BOOL;
	SendJIAOYAN_DATA:UINT;
	Judge_Xuhao:BOOL;
	Judge_Jiaoyan:BOOL;
	Ver_Output1:DWORD;
	Time_Minute_Left1:UINT;
	GPS_Signal_Intensity1:BYTE;
	VarCanGpsTongXunLockCommand_2:BOOL;
	send_data220_enable:BOOL;
	send_trig:R_TRIG;
	i_count:UINT;
	clear_zhiling:BOOL;
	tCounter:BYTE;
	CANI_Button_RecordClear11:BOOL;
	tCounter2:BYTE;
	
	
	CAN2_SEND_220:ifmRCAN.CAN_Tx;
	CAN2_SEND_2C0:ifmRCAN.CAN_Tx;
	CAN2_SEND_2E0:ifmRCAN.CAN_Tx;
	CAN2_SEND_200:ifmRCAN.CAN_Tx;
	CAN2_SEND_201:ifmRCAN.CAN_Tx;
	CAN2_SEND_202:ifmRCAN.CAN_Tx;
	CAN2_SEND_203:ifmRCAN.CAN_Tx;
	CAN2_SEND_204:ifmRCAN.CAN_Tx;
	CAN2_SEND_205:ifmRCAN.CAN_Tx;
	CAN2_SEND_206:ifmRCAN.CAN_Tx;
	CAN2_SEND_207:ifmRCAN.CAN_Tx;
	CAN2_SEND_20A:ifmRCAN.CAN_Tx;
	CAN2_SEND_20B:ifmRCAN.CAN_Tx;
	CAN2_SEND_20C:ifmRCAN.CAN_Tx;
	CAN2_SEND_20D:ifmRCAN.CAN_Tx;
	CAN2_SEND_20E:ifmRCAN.CAN_Tx;
	CAN2_SEND_211:ifmRCAN.CAN_Tx;
	CAN2_SEND_212:ifmRCAN.CAN_Tx;
	CAN2_SEND_213:ifmRCAN.CAN_Tx;
	CAN2_SEND_214:ifmRCAN.CAN_Tx;
	CAN2_SEND_215:ifmRCAN.CAN_Tx;
	CAN2_SEND_216:ifmRCAN.CAN_Tx;
	CAN2_SEND_217:ifmRCAN.CAN_Tx;
	CAN2_SEND_218:ifmRCAN.CAN_Tx;
	CAN2_SEND_2F0:ifmRCAN.CAN_Tx;
	CAN2_SEND_2FF:ifmRCAN.CAN_Tx;
	CAN2_SEND_280:ifmRCAN.CAN_Tx;
	CAN2_SEND_281:ifmRCAN.CAN_Tx;
	CAN2_SEND_282:ifmRCAN.CAN_Tx;
	CAN2_SEND_283:ifmRCAN.CAN_Tx;
	CAN2_SEND_284:ifmRCAN.CAN_Tx;
	CAN2_SEND_2B0:ifmRCAN.CAN_Tx;
	CAN2_SEND_2B1:ifmRCAN.CAN_Tx;
	CAN1_SEND_18FF0001:ifmRCAN.CAN_Tx;
	
	CAN2_RECE_GPS300:ifmRCAN.CAN_Rx;
	CAN2_RECE_GPS303:ifmRCAN.CAN_Rx;
	CAN2_RECE_GPS320:ifmRCAN.CAN_Rx;
	CAN2_RECE_GPS321:ifmRCAN.CAN_Rx;
	CAN2_RECE_GPS322:ifmRCAN.CAN_Rx;
	CAN2_RECE_GPS323:ifmRCAN.CAN_Rx;
	CAN2_RECE_GPS324:ifmRCAN.CAN_Rx;
	CAN2_RECE_GPS325:ifmRCAN.CAN_Rx;
	TIME_60s_3:TON;END_VAR

TIME_100ms(IN:=NOT TIME_100ms.Q,PT:=T#100MS);
TIME_500ms(IN:=NOT TIME_500ms.Q,PT:=T#500MS);
TIME_510ms(IN:=NOT TIME_510ms.Q,PT:=T#510MS);
TIME_520ms(IN:=NOT TIME_520ms.Q,PT:=T#520MS);
TIME_530ms(IN:=NOT TIME_530ms.Q,PT:=T#530MS);
TIME_1000ms(IN:=NOT TIME_1000ms.Q,PT:=T#1000MS);
TIME_1000ms_2(IN:=NOT TIME_1000ms_2.Q,PT:=T#1000MS);
TIME_10s(IN:=TRUE,PT:=T#10S);
TIME_5s(IN:=TRUE,PT:=T#5S);

(*控制器接受GPS数据*)
CAN2_RECE_GPS300(xEnable:=TRUE , eChannel:= 1, xExtended:= FALSE, aData=> receive_data300, udiID:= 16#300);
CAN2_RECE_GPS303(xEnable:=TRUE , eChannel:= 1, xExtended:= FALSE, aData=> receive_data303, udiID:= 16#303);
CAN2_RECE_GPS320(xEnable:=TRUE , eChannel:= 1, xExtended:= FALSE, aData=> receive_data320, udiID:= 16#320);
CAN2_RECE_GPS321(xEnable:=TRUE , eChannel:= 1, xExtended:= FALSE, aData=> receive_data321, udiID:= 16#321);
CAN2_RECE_GPS322(xEnable:=TRUE , eChannel:= 1, xExtended:= FALSE, aData=> receive_data322, udiID:= 16#322);
CAN2_RECE_GPS323(xEnable:=TRUE , eChannel:= 1, xExtended:= FALSE, aData=> receive_data323, udiID:= 16#323);
CAN2_RECE_GPS324(xEnable:=TRUE , eChannel:= 1, xExtended:= FALSE, aData=> receive_data324, udiID:= 16#324);
CAN2_RECE_GPS325(xEnable:=TRUE , eChannel:= 1, xExtended:= FALSE, aData=> receive_data325, udiID:= 16#325);


(*接收时间*)
		GPS_Time_bool:=USINT_TO_BOOL(receive_data303[0]);
		GPS_Time_Year:=receive_data303[1];
		GPS_Time_Month:=receive_data303[2];
		GPS_Time_Day:=receive_data303[3];
		GPS_Time_Hour:=receive_data303[4];
		GPS_Time_Minute:=receive_data303[5];
		GPS_Time_Second:=receive_data303[6];
		GPS_Signal_Intensity:=receive_data303[7];
GPS_Signal_Intensity1:=(105-GPS_Signal_Intensity)+128;
send_data18FF0001[0]:=UINT_TO_USINT(Time_Minute_Left MOD 256);
send_data18FF0001[1]:=UINT_TO_USINT(Time_Minute_Left / 256);
send_data18FF0001[2]:=PACK(B0:=VarCanNewGpsNoSignalLock_Warning OR VarCanNewGpsNoSignalLock_Warning2,
						   B1:=(VarGpsSystemLockedState_bool OR (VarCanGpsTongXunLockCommand AND VarGpsGlobalEnable)),
						   B2:=VarGpsSystemLockedState,B3:=0,
						   B4:=0,B5:=0,B6:=0,B7:=0);
send_data18FF0001[3]:=GPS_Signal_Intensity;
send_data18FF0001[4]:=0;
send_data18FF0001[5]:=0;
send_data18FF0001[6]:=0;
send_data18FF0001[7]:=0;
IF TIME_100ms.Q THEN
	CAN1_SEND_18FF0001(xEnable:= TRUE, eChannel:= 0, udiID:= 16#18FF0001, xExtended:=TRUE, usiDLC:=8 , aData:=send_data18FF0001);
END_IF

(*发送数据*)
send_data200[0]:=04;(**协议版本**)
send_data200[1]:=UINT_TO_USINT(0);(**硬件版本**)
send_data200[2]:=UINT_TO_USINT(0);(**软件版本**)
send_data200[3]:=UINT_TO_USINT(1);(**加密标识**)
send_data200[4]:=UINT_TO_USINT(0 MOD 256);(**控制器序列号**)
send_data200[5]:=UINT_TO_USINT(0 /256);
send_data200[6]:=UINT_TO_USINT(0 MOD 256);
send_data200[7]:=UINT_TO_USINT(0/256);

send_data201[3]:=INT_TO_USINT(255)-PACK(B0:=VarGpsSystemLockedState,B1:=VarCanGpsLockCommand_B,B2:=VarCanGpsLockCommand_C,
                      B3:=VarCanGpsLockCommand_D,B4:=VarCanGpsLockCommand_E,B5:=VarCanGpsKongZhiQiLockCommand,
                      B6:=VarCanGpsLockCommand_B1,B7:=VarCanGpsLockCommand_C1);
send_data201[2]:=INT_TO_USINT(255)-PACK(B0:=VarCanGpsLockCommand_D1,B1:=VarCanGpsLockCommand_E1,B2:=VarCanGpsBEIDONGLockCommand,
                      B3:=VarCanGpsYanShiLockCommand_Enable,B4:=VarCanGpsKaiGaiLockCommand_Enable,B5:=VarCanGpsTongXunLockCommand_Enable,
                      B6:=VarCanGpsBakaLockCommand_Enable,B7:=0);
send_data201[1]:=INT_TO_USINT(255)-PACK(B0:=VarCanGpsYanShiLockCommand,B1:=VarCanGpsKaiGaiLockCommand,B2:=VarCanGpsTongXunLockCommand,
                      B3:=VarCanGpsTianXianLockCommand,B4:=VarCanGpsTianXianLockCommand,B5:=VarGpsGlobalEnable,
                      B6:=VarGpsTempUnlockDoing,B7:=0);
send_data201[0]:=INT_TO_USINT(255)-PACK(B0:=0,B1:=0,B2:=0,
                      B3:=0,B4:=0,B5:=0,
                      B6:=0,B7:=0);
send_data201[7]:=INT_TO_USINT(255)-UDINT_TO_USINT((CANO_Accumu_Fuel MOD 65536) MOD 256);(**总油耗**)
send_data201[6]:=INT_TO_USINT(255)-UDINT_TO_USINT((CANO_Accumu_Fuel MOD 65536) /256);
send_data201[5]:=INT_TO_USINT(255)-UDINT_TO_USINT((CANO_Accumu_Fuel / 65536) MOD 256);
send_data201[4]:=INT_TO_USINT(255)-UDINT_TO_USINT((CANO_Accumu_Fuel / 65536)/256);

send_data202[3]:=INT_TO_USINT(255)-UDINT_TO_USINT((CANO_ACCMUDEPTH/100 MOD 65536) MOD 256);(**总油耗**)
send_data202[2]:=INT_TO_USINT(255)-UDINT_TO_USINT((CANO_ACCMUDEPTH/100 MOD 65536) /256);
send_data202[1]:=INT_TO_USINT(255)-UDINT_TO_USINT((CANO_ACCMUDEPTH/100 / 65536) MOD 256);
send_data202[0]:=INT_TO_USINT(255)-UDINT_TO_USINT((CANO_ACCMUDEPTH/100 / 65536)/256);
send_data202[4]:=INT_TO_USINT(255)-TO_USINT(CANO_water_tem);(**水温**)
send_data202[5]:=INT_TO_USINT(255)-UINT_TO_USINT(CANO_Hyd_Tem);(**油温**)
send_data202[6]:=INT_TO_USINT(255)-UINT_TO_USINT(CANO_FUEL_LEVEL);(**燃油液位**)
send_data202[7]:=INT_TO_USINT(255)-UINT_TO_USINT(CANO_Lub_Press);(**机油压力**)

send_data203[1]:=INT_TO_USINT(255)-UINT_TO_USINT((CANO_SPEED) MOD 256);(**发动机转速**)
send_data203[0]:=INT_TO_USINT(255)-UINT_TO_USINT((CANO_SPEED)/256);
send_data203[4]:=INT_TO_USINT(255)-UDINT_TO_USINT((CANO_engine_hour_h ) MOD 256);(**累计工作小时**)
send_data203[3]:=INT_TO_USINT(255)-UDINT_TO_USINT((CANO_engine_hour_h ) /256);(**累计工作小时**)
send_data203[2]:=INT_TO_USINT(255)-UDINT_TO_USINT((CANO_engine_hour_h / 65536) MOD 256);;(**累计工作小时**)
send_data203[5]:=INT_TO_USINT(255)-UDINT_TO_USINT(CANO_engine_hour_m MOD 60 );(**工作分钟**)
send_data203[7]:=INT_TO_USINT(255)-UINT_TO_USINT((FuelMomentary) MOD 256);;(**瞬间油耗**)
send_data203[6]:=INT_TO_USINT(255)-UINT_TO_USINT((FuelMomentary)/256);

send_data204[0]:=INT_TO_USINT(255)-UINT_TO_USINT(CANO_PilotPressure/10);(**先导压力**)
send_data204[1]:=INT_TO_USINT(255)-UINT_TO_USINT(Codes_FMI_1);(**FMI**)
send_data204[3]:=INT_TO_USINT(255)-UDINT_TO_USINT(Codes_SPN_1 MOD 256);(**SPN**)
send_data204[2]:=INT_TO_USINT(255)-UDINT_TO_USINT(Codes_SPN_1/256);
send_data204[4]:=INT_TO_USINT(255)-UINT_TO_USINT(VarMastLimitState);(**限位模式,1为上限位，2为下限位**)
send_data204[5]:=INT_TO_USINT(255)-PACK(B0:=0,(**快放模式*)
					  B1:=DOH_Y56,(**主卷浮动*)
 					  B2:=DOH_Y51,(**先导使能**)
 					  B3:=CANO_RotationModle,(**回转模式*)
 					  B4:=VarMastAutoEnable,(**调平模式*)
 					  B5:=CANI_Button_DepthClear,(**深度清零**)
 					  B6:=0,
 					  B7:=0);(****)
send_data204[6]:=INT_TO_BYTE(255)-PACK(B0:=CANO_TooLow_OilPress,(**机油压力低报警**)
					  B1:=CANO_TooHigh_WaterTem,(**水温高报警**)
 					  B2:=CANO_TooHigh_HydOilTem,(**液压油温高报警**)
 					  B3:=CANO_TooLow_FUEL_LEVEL,(**燃油液位低报警**)
 					  B4:=CANO_TooLow_BatteryVol,(**电瓶电压低报警**)
 					  B5:=0,
 					  B6:=0,(**无**)
 					  B7:=DIH_SP4);(**滤芯堵塞报警**)
send_data204[7]:=INT_TO_BYTE(255)-PACK(B0:=DIH_SQ8,(**重锤上限位**)
					  B1:=0,(**触底保护**)
 					  B2:=0,(****)
 					  B3:=0,(****)
 					  B4:=0,(****)
 					  B5:=0,(****)
 					  B6:=0,(****)
 					  B7:=0);(****)
send_data205[3]:=INT_TO_BYTE(255)-UDINT_TO_USINT((0 MOD 65536) MOD 256);(**施工槽号**)
send_data205[2]:=INT_TO_BYTE(255)-UDINT_TO_USINT((0 MOD 65536) /256);
send_data205[1]:=INT_TO_BYTE(255)-UDINT_TO_USINT((0 / 65536) MOD 256);
send_data205[0]:=INT_TO_BYTE(255)-UDINT_TO_USINT((0 / 65536)/256);
send_data205[5]:=INT_TO_BYTE(255)-UINT_TO_USINT(0 MOD 256);(**槽宽**)
send_data205[4]:=INT_TO_BYTE(255)-UINT_TO_USINT(0/256);
send_data205[7]:=INT_TO_BYTE(255)-UINT_TO_USINT(CANO_DEPTH MOD 256);(**当前槽深**)
send_data205[6]:=INT_TO_BYTE(255)-UINT_TO_USINT(CANO_DEPTH/256);

send_data206[1]:=INT_TO_BYTE(255)-UINT_TO_USINT(CANO_ANGLE_X MOD 256);(**倾角X**)
send_data206[0]:=INT_TO_BYTE(255)-UINT_TO_USINT(CANO_ANGLE_X/256);
send_data206[3]:=INT_TO_BYTE(255)-UINT_TO_USINT(CANO_ANGLE_Y MOD 256);(**倾角Y**)
send_data206[2]:=INT_TO_BYTE(255)-UINT_TO_USINT(CANO_ANGLE_Y/256);
send_data206[5]:=INT_TO_BYTE(255)-UINT_TO_USINT(CANO_MainWinch_Speed MOD 256);(**主卷速度**)
send_data206[4]:=INT_TO_BYTE(255)-UINT_TO_USINT(CANO_MainWinch_Speed/256);
send_data206[7]:=INT_TO_BYTE(255)-UINT_TO_USINT(CANO_PowerHeadTorque MOD 256);(**动力头扭矩*)
send_data206[6]:=INT_TO_BYTE(255)-UINT_TO_USINT(CANO_PowerHeadTorque/256);(****)

send_data207[0]:=INT_TO_BYTE(255)-UINT_TO_USINT(CANO_PowerHeadSpeed);(**动力头转速*)
send_data207[1]:=INT_TO_BYTE(255)-UINT_TO_USINT(CANO_DonglitouPressure/10);(**动力头压力*)
send_data207[2]:=INT_TO_BYTE(255)-UINT_TO_USINT(CANO_JiayaPressure /10);(**推进压力*)
send_data207[3]:=INT_TO_BYTE(255)-UINT_TO_USINT(CANO_ZhuJuanPressure/10);(**主卷扬压力*)
send_data207[4]:=INT_TO_BYTE(255)-UINT_TO_USINT(0 MOD 256);
send_data207[4]:=INT_TO_BYTE(255)-UINT_TO_USINT(0/256);
send_data207[7]:=INT_TO_BYTE(255)-UINT_TO_USINT(0 MOD 256);
send_data207[6]:=INT_TO_BYTE(255)-UINT_TO_USINT(0/256);

send_data20A[1]:=INT_TO_BYTE(255)-UINT_TO_USINT(PAR_Circle1 MOD 256);(**转盘外层直径**)
send_data20A[0]:=INT_TO_BYTE(255)-UINT_TO_USINT(PAR_Circle1/256);
send_data20A[3]:=INT_TO_BYTE(255)-UINT_TO_USINT(PAR_Circle2 MOD 256);(**转盘内层直径*)
send_data20A[2]:=INT_TO_BYTE(255)-UINT_TO_USINT(PAR_Circle2/256);
send_data20A[5]:=INT_TO_BYTE(255)-UINT_TO_USINT(PAR_ControlValue MOD 256);(**步长值*)
send_data20A[4]:=INT_TO_BYTE(255)-UINT_TO_USINT(PAR_ControlValue/256);
send_data20A[6]:=INT_TO_BYTE(255)-UINT_TO_USINT(PAR_Quanshu);(**外层圈数*)
send_data20A[7]:=INT_TO_BYTE(255)-UINT_TO_USINT(0);

send_data20B[1]:=INT_TO_BYTE(255)-UINT_TO_USINT(PAR_Y27_PosFull MOD 256);(**阀A正向最大电流*)
send_data20B[0]:=INT_TO_BYTE(255)-UINT_TO_USINT(PAR_Y27_PosFull/256);
send_data20B[3]:=INT_TO_BYTE(255)-UINT_TO_USINT(PAR_Y27_NegFull MOD 256);(**阀A正向最小电流*)
send_data20B[2]:=INT_TO_BYTE(255)-UINT_TO_USINT(PAR_Y27_NegFull/256);
send_data20B[5]:=INT_TO_BYTE(255)-UINT_TO_USINT(PAR_Y28_PosFull MOD 256);(**阀A逆向最大电流*)
send_data20B[4]:=INT_TO_BYTE(255)-UINT_TO_USINT(PAR_Y28_PosFull/256);
send_data20B[7]:=INT_TO_BYTE(255)-UINT_TO_USINT(PAR_Y28_NegFull MOD 256);(**阀A逆向最小电流*)
send_data20B[6]:=INT_TO_BYTE(255)-UINT_TO_USINT(PAR_Y28_NegFull/256);

send_data20C[1]:=INT_TO_BYTE(255)-UINT_TO_USINT(PAR_Y29_PosFull MOD 256);(**阀B正向最大电流*)
send_data20C[0]:=INT_TO_BYTE(255)-UINT_TO_USINT(PAR_Y29_PosFull/256);
send_data20C[3]:=INT_TO_BYTE(255)-UINT_TO_USINT(PAR_Y29_NegFull MOD 256);(**阀B正向最小电流*)
send_data20C[2]:=INT_TO_BYTE(255)-UINT_TO_USINT(PAR_Y29_NegFull/256);
send_data20C[4]:=INT_TO_BYTE(255)-UINT_TO_USINT(PAR_WarnFuelLevel_Low);(**燃油低液位*)
send_data20C[5]:=INT_TO_BYTE(255)-UINT_TO_USINT(PAR_WarnHydOilTem_High);(*液压油温高*)
send_data20C[6]:=INT_TO_BYTE(255)-UINT_TO_USINT(PAR_WarnOilPress_Low );(**机油压力低*)
send_data20C[7]:=INT_TO_BYTE(255)-UINT_TO_USINT(0/256);


send_data20D[1]:=INT_TO_BYTE(255)-UINT_TO_USINT(PAR_HydOilPilotPress_NegFull MOD 256);(**压力下限**)
send_data20D[0]:=INT_TO_BYTE(255)-UINT_TO_USINT(PAR_HydOilPilotPress_NegFull/256);
send_data20D[3]:=INT_TO_BYTE(255)-UINT_TO_USINT(PAR_HydOilPress_PosFull MOD 256);(**压力上限**)
send_data20D[2]:=INT_TO_BYTE(255)-UINT_TO_USINT(PAR_HydOilPress_PosFull/256);
send_data20D[5]:=INT_TO_BYTE(255)-UINT_TO_USINT(PAR_SpeedLow_Idling MOD 256);(**发动机低怠速**)
send_data20D[4]:=INT_TO_BYTE(255)-UINT_TO_USINT(PAR_SpeedLow_Idling/256);
send_data20D[7]:=INT_TO_BYTE(255)-UINT_TO_USINT(PAR_SpeedHigh_Idling MOD 256);(**发动机高怠速**)
send_data20D[6]:=INT_TO_BYTE(255)-UINT_TO_USINT(PAR_SpeedHigh_Idling/256);

send_data20E[1]:=INT_TO_BYTE(255)-UINT_TO_USINT(PAR_Y30_PosFull MOD 256);(**阀B逆向最大电流*)
send_data20E[0]:=INT_TO_BYTE(255)-UINT_TO_USINT(PAR_Y30_PosFull/256);
send_data20E[3]:=INT_TO_BYTE(255)-UINT_TO_USINT(PAR_Y30_NegFull MOD 256);(**阀A逆向最小电流*)
send_data20E[2]:=INT_TO_BYTE(255)-UINT_TO_USINT(PAR_Y30_NegFull/256);
send_data20E[4]:=INT_TO_BYTE(255)-UINT_TO_USINT(0);
send_data20E[5]:=INT_TO_BYTE(255)-UINT_TO_USINT(0);
send_data20E[6]:=INT_TO_BYTE(255)-UINT_TO_USINT(0 );
send_data20E[7]:=INT_TO_BYTE(255)-UINT_TO_USINT(0/256);

send_data211[1]:=INT_TO_BYTE(255)-UINT_TO_USINT(CANI_JOYX_L MOD 256);(****)
send_data211[0]:=INT_TO_BYTE(255)-UINT_TO_USINT(CANI_JOYX_L/256);
send_data211[3]:=INT_TO_BYTE(255)-UINT_TO_USINT(CANI_JOYY_L MOD 256);(****)
send_data211[2]:=INT_TO_BYTE(255)-UINT_TO_USINT(CANI_JOYY_L/256);
send_data211[5]:=INT_TO_BYTE(255)-UINT_TO_USINT(CANI_JOYX_R MOD 256);(****)
send_data211[4]:=INT_TO_BYTE(255)-UINT_TO_USINT(CANI_JOYX_R/256);
send_data211[7]:=INT_TO_BYTE(255)-UINT_TO_USINT(CANI_JOYY_R MOD 256);(****)
send_data211[6]:=INT_TO_BYTE(255)-UINT_TO_USINT(CANI_JOYY_R/256);

send_data212[1]:=INT_TO_BYTE(255)-UINT_TO_USINT(CANI_JOY_Jiao_L MOD 256);(****)
send_data212[0]:=INT_TO_BYTE(255)-UINT_TO_USINT(CANI_JOY_Jiao_L/256);
send_data212[3]:=INT_TO_BYTE(255)-UINT_TO_USINT(CANI_JOY_Jiao_R MOD 256);(****)
send_data212[2]:=INT_TO_BYTE(255)-UINT_TO_USINT(CANI_JOY_Jiao_R/256);
send_data212[5]:=INT_TO_BYTE(255)-UINT_TO_USINT(PWM_Y1 MOD 256);(****)
send_data212[4]:=INT_TO_BYTE(255)-UINT_TO_USINT(PWM_Y1/256);
send_data212[7]:=INT_TO_BYTE(255)-UINT_TO_USINT(PWM_Y2 MOD 256);(****)
send_data212[6]:=INT_TO_BYTE(255)-UINT_TO_USINT(PWM_Y2/256);

send_data213[1]:=INT_TO_BYTE(255)-UINT_TO_USINT(PWM_Y7 MOD 256);(****)
send_data213[0]:=INT_TO_BYTE(255)-UINT_TO_USINT(PWM_Y7/256);
send_data213[3]:=INT_TO_BYTE(255)-UINT_TO_USINT(PWM_Y8 MOD 256);(****)
send_data213[2]:=INT_TO_BYTE(255)-UINT_TO_USINT(PWM_Y8/256);
send_data213[5]:=INT_TO_BYTE(255)-UINT_TO_USINT(PWM_Y9 MOD 256);(****)
send_data213[4]:=INT_TO_BYTE(255)-UINT_TO_USINT(PWM_Y9/256);
send_data213[7]:=INT_TO_BYTE(255)-UINT_TO_USINT(PWM_Y10 MOD 256);(****)
send_data213[6]:=INT_TO_BYTE(255)-UINT_TO_USINT(PWM_Y10/256);

send_data214[1]:=INT_TO_BYTE(255)-UINT_TO_USINT(PWM_Y11 MOD 256);(****)
send_data214[0]:=INT_TO_BYTE(255)-UINT_TO_USINT(PWM_Y11/256);
send_data214[3]:=INT_TO_BYTE(255)-UINT_TO_USINT(PWM_Y12 MOD 256);(****)
send_data214[2]:=INT_TO_BYTE(255)-UINT_TO_USINT(PWM_Y12/256);
send_data214[5]:=INT_TO_BYTE(255)-UINT_TO_USINT(PWM_Y13 MOD 256);(****)
send_data214[4]:=INT_TO_BYTE(255)-UINT_TO_USINT(PWM_Y13/256);
send_data214[7]:=INT_TO_BYTE(255)-UINT_TO_USINT(PWM_Y14 MOD 256);(****)
send_data214[6]:=INT_TO_BYTE(255)-UINT_TO_USINT(PWM_Y14/256);

send_data215[1]:=INT_TO_BYTE(255)-UINT_TO_USINT(PWM_Y60 MOD 256);(****)
send_data215[0]:=INT_TO_BYTE(255)-UINT_TO_USINT(PWM_Y60/256);
send_data215[3]:=INT_TO_BYTE(255)-UINT_TO_USINT(PWM_Y61 MOD 256);(****)
send_data215[2]:=INT_TO_BYTE(255)-UINT_TO_USINT(PWM_Y61/256);
send_data215[5]:=INT_TO_BYTE(255)-UINT_TO_USINT(PWM_Y23 MOD 256);(****)
send_data215[4]:=INT_TO_BYTE(255)-UINT_TO_USINT(PWM_Y23/256);
send_data215[7]:=INT_TO_BYTE(255)-UINT_TO_USINT(PWM_Y24 MOD 256);(****)
send_data215[6]:=INT_TO_BYTE(255)-UINT_TO_USINT(PWM_Y24/256);

send_data216[1]:=INT_TO_BYTE(255)-UINT_TO_USINT(PWM_Y21 MOD 256);(****)
send_data216[0]:=INT_TO_BYTE(255)-UINT_TO_USINT(PWM_Y21/256);
send_data216[3]:=INT_TO_BYTE(255)-UINT_TO_USINT(PWM_Y22 MOD 256);(****)
send_data216[2]:=INT_TO_BYTE(255)-UINT_TO_USINT(PWM_Y22/256);
send_data216[5]:=INT_TO_BYTE(255)-UINT_TO_USINT(PWM_Y5 MOD 256);(****)
send_data216[4]:=INT_TO_BYTE(255)-UINT_TO_USINT(PWM_Y5/256);
send_data216[7]:=INT_TO_BYTE(255)-UINT_TO_USINT(PWM_Y6 MOD 256);(****)
send_data216[6]:=INT_TO_BYTE(255)-UINT_TO_USINT(PWM_Y6/256);

send_data217[1]:=INT_TO_BYTE(255)-UINT_TO_USINT(PWM_Y34 MOD 256);(****)
send_data217[0]:=INT_TO_BYTE(255)-UINT_TO_USINT(PWM_Y34/256);
send_data217[3]:=INT_TO_BYTE(255)-UINT_TO_USINT(PWM_Y33 MOD 256);(****)
send_data217[2]:=INT_TO_BYTE(255)-UINT_TO_USINT(PWM_Y33/256);
send_data217[5]:=INT_TO_BYTE(255)-UINT_TO_USINT(PWM_Y39 MOD 256);(****)
send_data217[4]:=INT_TO_BYTE(255)-UINT_TO_USINT(PWM_Y39/256);
send_data217[7]:=INT_TO_BYTE(255)-UINT_TO_USINT(PWM_Y40 MOD 256);(****)
send_data217[6]:=INT_TO_BYTE(255)-UINT_TO_USINT(PWM_Y40 MOD 256);(****)


send_data218[0]:=INT_TO_BYTE(255)-PACK(B0:=CANI_JOY_SB1,(**重锤上限位**)
					  B1:=CANI_JOY_SB2,(**触底保护**)
 					  B2:=CANI_JOY_SB3,(****)
 					  B3:=CANI_JOY_SB4,(****)
 					  B4:=CANI_JOY_SB5,(****)
 					  B5:=CANI_JOY_SB6,(****)
 					  B6:=CANI_JOY_SB7,(****)
 					  B7:=0);(****)
send_data218[1]:=0;
send_data218[3]:=INT_TO_BYTE(255)-UINT_TO_USINT(DI_LHandle_SB4_UINT MOD 256);(****)
send_data218[2]:=INT_TO_BYTE(255)-UINT_TO_USINT(DI_LHandle_SB4_UINT/256);
send_data218[5]:=INT_TO_BYTE(255)-UINT_TO_USINT(DI_RHandle_SB7_UINT MOD 256);(****)
send_data218[4]:=INT_TO_BYTE(255)-UINT_TO_USINT(DI_RHandle_SB7_UINT/256);
send_data218[7]:=0;(****)
send_data218[6]:=0;(****)

(*接收到平台的请求读指令后，发送无信号锁车时间给平台*)
IF (receive_data324[3]=16#03 AND receive_data324[4]=16#E8)THEN
	send_data220_enable:=TRUE;
END_IF
IF send_data220_enable THEN
	send_data220[1]:=INT_TO_BYTE(255)-UINT_TO_USINT(1000 MOD 256);(****)
	send_data220[0]:=INT_TO_BYTE(255)-UINT_TO_USINT(1000/256);
	send_data220[3]:=INT_TO_BYTE(255)-UINT_TO_USINT((VarCanGpsYanShiLockCommand_time ) MOD 256);(****)
	send_data220[2]:=INT_TO_BYTE(255)-UINT_TO_USINT((VarCanGpsYanShiLockCommand_time )/256);
	send_data220[5]:=INT_TO_BYTE(255)-UINT_TO_USINT((0) MOD 256);(****)
	send_data220[4]:=INT_TO_BYTE(255)-UINT_TO_USINT((0) / 256);
	send_data220[7]:=INT_TO_BYTE(255)-UINT_TO_USINT(0 MOD 256);(****)
	send_data220[6]:=INT_TO_BYTE(255)-UINT_TO_USINT(0 MOD 256);(****)
	CAN2_SEND_220(xEnable:= TRUE, eChannel:= 1, udiID:= 16#220, xExtended:=FALSE, usiDLC:=8 , aData:=send_data220);
END_IF
(*接收到平台的请求写指令后，修改无信号锁车时间*)
IF (receive_data325[3]=16#01 ) THEN
	VarCanGpsYanShiLockCommand_time:=receive_data325[5]+receive_data325[4]*256;
END_IF

send_data280[0]:=UINT_TO_USINT(1);(****)
send_data280[2]:=UINT_TO_USINT(count MOD 256);
send_data280[1]:=UINT_TO_USINT(count/256);(**发送次数**)
send_data280[3]:=UINT_TO_USINT(0);
send_data280[5]:=UINT_TO_USINT(CANO_PowerHeadTorque MOD 256);(**动力头扭矩**)
send_data280[4]:=UINT_TO_USINT(CANO_PowerHeadTorque/256);
send_data280[6]:=UINT_TO_USINT(CANO_PowerHeadSpeed);(**动力头转速**)
send_data280[7]:=BOOL_TO_USINT(0);(*快放模式*)

send_data281[0]:=UINT_TO_USINT(2);(****)
send_data281[2]:=UINT_TO_USINT(CANO_ANGLE_X MOD 256);
send_data281[1]:=UINT_TO_USINT(CANO_ANGLE_X/256);(****)
send_data281[4]:=UINT_TO_USINT(CANO_ANGLE_Y MOD 256);
send_data281[3]:=UINT_TO_USINT(CANO_ANGLE_Y / 256);(****)
send_data281[5]:=UINT_TO_USINT(CANO_DonglitouPressure/10);
send_data281[6]:=UINT_TO_USINT(CANO_JiayaPressure / 10);(****)
send_data281[7]:=UINT_TO_USINT(CANO_ZhuJuanPressure/10);

send_data282[0]:=UINT_TO_USINT(3);(****)
send_data282[1]:=UINT_TO_USINT(0 MOD 256);
send_data282[5]:=UDINT_TO_USINT((PileNumble MOD 65536) MOD 256);(**桩号*)
send_data282[4]:=UDINT_TO_USINT((PileNumble MOD 65536) /256);
send_data282[3]:=UDINT_TO_USINT((PileNumble / 65536) MOD 256);
send_data282[2]:=UDINT_TO_USINT((PileNumble / 65536)/256);
send_data282[7]:=UINT_TO_USINT(PileDiameter MOD 256);(****)
send_data282[6]:=UINT_TO_USINT(PileDiameter/256);

send_data283[0]:=UINT_TO_USINT(4);(****)
send_data283[1]:=UINT_TO_USINT(0/256);
send_data283[3]:=UINT_TO_USINT(CANO_DEPTH MOD 256);(****)
send_data283[2]:=UINT_TO_USINT(CANO_DEPTH/256);
send_data283[5]:=UINT_TO_USINT(CANO_X_PIANYIZHI MOD 256);
send_data283[4]:=UINT_TO_USINT(CANO_X_PIANYIZHI/256);
send_data283[7]:=UINT_TO_USINT(CANO_Y_PIANYIZHI MOD 256);(****)
send_data283[6]:=UINT_TO_USINT(CANO_Y_PIANYIZHI/256);

send_data284[0]:=UINT_TO_USINT(5);(****)
send_data284[2]:=UINT_TO_USINT(CANO_MainWinch_Speed MOD 256);(****)
send_data284[1]:=UINT_TO_USINT(CANO_MainWinch_Speed / 256);(****)
send_data284[2]:=UINT_TO_USINT(0/256);
send_data284[5]:=UINT_TO_USINT(0 MOD 256);(****)
send_data284[4]:=UINT_TO_USINT(0/256);
send_data284[7]:=UINT_TO_USINT(0 MOD 256);(****)
send_data284[6]:=UINT_TO_USINT(0/256);

send_data2B0[0]:=UINT_TO_USINT(SaveEngineMode);(**节能模式**)
send_data2B0[1].0:=SaveEngineState;
send_data2B0[1].1:=CANO_SensorError_PAtomsPre;
send_data2B0[1].2:=CANO_SensorError_PAcPre;
send_data2B0[1].3:=CANO_SensorError_PM2;
send_data2B0[1].4:=CANO_SensorError_PM1;
send_data2B0[2]:=UINT_TO_USINT(GVL_SaveEngine.AI_PAtomsPre / 256);
send_data2B0[3]:=UINT_TO_USINT(GVL_SaveEngine.AI_PAtomsPre MOD 256);
send_data2B0[4].0:=1;
send_data2B0[4].1:=1;
send_data2B0[4].2:=1;
send_data2B0[4].3:=1;
send_data2B0[4].4:=1;
send_data2B0[5]:=20;
send_data2B0[6]:=1;
send_data2B0[7]:=1;

send_data2B1[0]:=1;
send_data2B1[1]:=1;
send_data2B1[2]:=1;
send_data2B1[3]:=2;
send_data2B1[4]:=1;
send_data2B1[5]:=3;
send_data2B1[6]:=1;
send_data2B1[7]:=4;

(*向平台发送清零指令*)
send_data2C0[1]:=UINT_TO_USINT(100 MOD 256);(****)
send_data2C0[0]:=UINT_TO_USINT(100/256);
send_data2C0[2]:=UINT_TO_USINT(0 MOD 256);(****)
send_data2C0[3]:=PACK(B0:=1,B1:=0,B2:=0,B3:=0,B4:=0,B5:=0,B6:=0,B7:=0);
send_data2C0[4]:=UINT_TO_USINT(0 MOD 256);(****)
send_data2C0[5]:=UINT_TO_USINT(0/256);
send_data2C0[6]:=UINT_TO_USINT(0 MOD 256);(****)
send_data2C0[7]:=UINT_TO_USINT(0/256);
clear_trig(CLK:=CANI_Button_RecordClear1);
IF(clear_trig.Q)THEN
	clear_zhiling:=TRUE;
END_IF
IF clear_zhiling THEN
	IF(tCounter<3)THEN
		IF(TIME_100ms.Q)THEN
			CAN2_SEND_2C0(xEnable:= TRUE, eChannel:= 1, udiID:= 16#2C0, xExtended:=FALSE, usiDLC:=8 , aData:=send_data2C0);
			tCounter := tCounter + 1;
		END_IF
	ELSE
		tCounter:=0;
		clear_zhiling:=FALSE;
	END_IF					
END_IF
CLEAR_Feedback:=BYTE_TO_BOOL(receive_data323[5] AND 2#00000001);(*平台反馈清零成功*)
SN_323_Feedback2C0:=receive_data323[3]*256+receive_data323[4];
IF(CLEAR_Feedback) AND (SN_323_Feedback2C0=100)THEN
	CANI_Button_RecordClear11:=TRUE;
ELSE
	CANI_Button_RecordClear11:=FALSE;
END_IF

	IF(tCounter2<20  AND  CANI_Button_RecordClear11 )THEN
		IF(TIME_510ms.Q)THEN
			tCounter2:=tCounter2+1;
			CANI_Button_RecordClear:=TRUE;
		END_IF
	ELSE
		CANI_Button_RecordClear:=FALSE;
	END_IF

	IF CANI_Button_RecordClear1 THEN
		CANI_Button_RecordClear:=TRUE;
	END_IF

(**********清零************)
(***********清零指令反馈,0x323,上升沿出发一次只发一条，避免连续发送多条***********)
(*清零按下按钮，需等待3秒，控制器需收到平台反馈清零成功消息方可执行清零指令
，清零成功后，如果还需清零，需断电后开电才能执行下一次清零操作*)
(*IF	clear_trig.Q  THEN
	Cal_Clear02:=TRUE;
	i_count:=i_count+1;
END_IF

IF Cal_Clear02 THEN
	Cal_Clear01:=Cal_Clear01+1;
END_IF

IF Cal_Clear01=40 THEN
	Cal_Clear02:=FALSE;
	Cal_Clear01:=0;
	Cal_Clear03:=TRUE;
	CLEAR_2C0_SN:=count;(*发送给2C0的清零指令序列号*)
ELSE
	Cal_Clear03:=FALSE;
END_IF

CLEAR_Feedback:=BYTE_TO_BOOL(receive_data323[5] AND 2#00000001);(*平台反馈清零成功*)

clear_trig01(CLK:=CLEAR_Feedback);

IF	clear_trig01.Q THEN
	CANI_Button_Record_Result_TRIG:=TRUE;
END_IF

IF CANI_Button_Record_Result_TRIG THEN
	Result_TRIG:=Result_TRIG+1;
END_IF

IF Result_TRIG>1000 THEN
	Result_TRIG:=0;
	CANI_Button_Record_Result_TRIG:=FALSE;
END_IF

SN_323_Feedback2C0:=receive_data323[3]*256+receive_data323[4];

IF	CLEAR_2C0_SN=SN_323_Feedback2C0 AND CANI_Button_Record_Result_TRIG THEN
	CANI_Button_RecordClear:=TRUE;
	CANI_Button_RecordClear1:=FALSE;
ELSE
	CANI_Button_RecordClear:=FALSE;
END_IF*)

(*应答*)
SN_321:=receive_data321[0]*256+receive_data321[1];
SN_322:=receive_data322[0]*256+receive_data322[1];
SN_323:=receive_data323[0]*256+receive_data323[1];
SN_324:=receive_data324[0]*256+receive_data324[1];
SN_325:=receive_data325[0]*256+receive_data325[1];
VarCANGPSYINGDAREC_ID:=receive_data320[1]+receive_data320[0]*256;
VarCANGPSYINGDAREC_DATA:=receive_data320[3]+receive_data320[2]*256;

IF(CAN2_RECE_GPS321.uiAvailable<>0)THEN
	VarCANGPSYINGDASEND_ID:=801;
	VarCANGPSYINGDASEND_DATA:=SN_321;
ELSIF(CAN2_RECE_GPS322.uiAvailable<>0)THEN
	VarCANGPSYINGDASEND_ID:=802;
	VarCANGPSYINGDASEND_DATA:=SN_322;
ELSIF(CAN2_RECE_GPS323.uiAvailable<>0)THEN
	VarCANGPSYINGDASEND_ID:=803;
	VarCANGPSYINGDASEND_DATA:=SN_323;
ELSIF(CAN2_RECE_GPS324.uiAvailable<>0)THEN
	VarCANGPSYINGDASEND_ID:=804;
	VarCANGPSYINGDASEND_DATA:=SN_324;
ELSIF(CAN2_RECE_GPS325.uiAvailable<>0)THEN
	VarCANGPSYINGDASEND_ID:=805;
	VarCANGPSYINGDASEND_DATA:=SN_325;
END_IF

send_data2E0[1]:=UINT_TO_USINT(VarCANGPSYINGDASEND_ID MOD 256);(****)
send_data2E0[0]:=UINT_TO_USINT(VarCANGPSYINGDASEND_ID/256);
send_data2E0[3]:=UINT_TO_USINT(VarCANGPSYINGDASEND_DATA MOD 256);(****)
send_data2E0[2]:=UINT_TO_USINT(VarCANGPSYINGDASEND_DATA/256);
send_data2E0[4]:=UINT_TO_USINT(0 MOD 256);(****)
send_data2E0[5]:=UINT_TO_USINT(0/256);
send_data2E0[6]:=UINT_TO_USINT(0 MOD 256);(****)
send_data2E0[7]:=UINT_TO_USINT(0/256);

IF(CAN2_RECE_GPS321.uiAvailable<>0)THEN
	CAN2_SEND_2E0(xEnable:= TRUE, eChannel:= 1, udiID:= 16#2E0, xExtended:=FALSE, usiDLC:=8 , aData:=send_data2E0);
ELSIF(CAN2_RECE_GPS322.uiAvailable<>0)THEN
	CAN2_SEND_2E0(xEnable:= TRUE, eChannel:= 1, udiID:= 16#2E0, xExtended:=FALSE, usiDLC:=8 , aData:=send_data2E0);	
ELSIF(CAN2_RECE_GPS323.uiAvailable<>0)THEN
	CAN2_SEND_2E0(xEnable:= TRUE, eChannel:= 1, udiID:= 16#2E0, xExtended:=FALSE, usiDLC:=8 , aData:=send_data2E0);
ELSIF(CAN2_RECE_GPS324.uiAvailable<>0)THEN
	CAN2_SEND_2E0(xEnable:= TRUE, eChannel:= 1, udiID:= 16#2E0, xExtended:=FALSE, usiDLC:=8 , aData:=send_data2E0);	
ELSIF(CAN2_RECE_GPS325.uiAvailable<>0)THEN
	CAN2_SEND_2E0(xEnable:= TRUE, eChannel:= 1, udiID:= 16#2E0, xExtended:=FALSE, usiDLC:=8 , aData:=send_data2E0);
END_IF

send_data2F0[0]:=UINT_TO_USINT(CANO_FUEL_LEVEL );(****)
send_data2F0[1]:=16#FF;
send_data2F0[2]:=16#FF;(****)
send_data2F0[2]:=16#FF;
send_data2F0[4]:=16#FF;(****)
send_data2F0[5]:=16#FF;
send_data2F0[6]:=16#FF;(****)
send_data2F0[7]:=16#FF;





//GPS锁车
(*300数据*)
VarCanGpsJIAOYANNUM:=receive_data300[1]+receive_data300[0]*256;
VarCanGpsJIAOYANMA:=receive_data300[3]+receive_data300[2]*256;
VarCanNewGpsManufacturers:=receive_data300[4];
VarCanNewGpsVersion:=receive_data300[5];
STATE_Satellite:=BYTE_TO_BOOL(receive_data300[7] AND 2#00000001);(*BYTE6/Bit0/卫星定位状态，0未定位，1已定位*)
STATE_ACC:=BYTE_TO_BOOL(receive_data300[7] AND 2#00000010);(*BYTE6/Bit1/ACC状态，0关，1开*)
STATE_WarnConnection:=BYTE_TO_BOOL(receive_data300[7] AND 2#00000100);(*BYTE6/Bit2/1，控制器与GPS通讯中断报警*)
STATE_WarnPoweroff:=BYTE_TO_BOOL(receive_data300[7] AND 2#00001000);(*BYTE6/Bit3/1，GPS断电报警*)
STATE_WarnPowerlow:=BYTE_TO_BOOL(receive_data300[7] AND 2#00010000);(*BYTE6/Bit4/1，GPS外部电源低电压报警*)
STATE_WarnModuleoff:=BYTE_TO_BOOL(receive_data300[7] AND 2#00100000);(*BYTE6/Bit5/1，GPS模块发生故障*)
STATE_WarnTIANXIANoff:=BYTE_TO_BOOL(receive_data300[7] AND 2#01000000);(*BYTE6/Bit6/1，GPS天线未接或被剪断*)
STATE_WarnPowerProtect:=BYTE_TO_BOOL(receive_data300[7] AND 2#10000000);(*BYTE6/Bit7/1，低电压保护状态*)

STATE_WarnKAIGAI:=BYTE_TO_BOOL(receive_data300[6] AND 2#00000001);(*BYTE7/Bit0/1，开盖报警*)
STATE_WarnBAKA:=BYTE_TO_BOOL(receive_data300[6] AND 2#00000010);(*BYTE7/Bit1/1，拔卡报警*)
IF TIME_10s.Q THEN
	STATE_Promoteconnect:=BYTE_TO_BOOL(receive_data300[6] AND 2#00000100);(*BYTE7/Bit2/1，与远程平台连接正常，0异常*)
END_IF
STATE_MASTERSleep:=BYTE_TO_BOOL(receive_data300[6] AND 2#00001000);(*BYTE7/Bit3/1，主电休眠状态*)
STATE_BACKUPSleep:=BYTE_TO_BOOL(receive_data300[6] AND 2#00010000);(*BYTE7/Bit4/1，备电休眠状态*)
(*GPS出现报警*)
(*IF	(*STATE_WarnConnection OR STATE_WarnPoweroff OR STATE_WarnPowerlow OR STATE_WarnModuleoff
	OR*) STATE_WarnTIANXIANoff OR STATE_WarnPowerProtect OR STATE_WarnKAIGAI OR STATE_WarnBAKA THEN
	STATE_WARN:=TRUE;
ELSE
	STATE_WARN:=FALSE;
END_IF*)
(*锁车*)
(*主控制器锁车*)
	IF VarCanGpsenableALLLockCommand THEN
		IF(BYTE_TO_BOOL(receive_data322[3] AND 2#00000001) )THEN
			VarCanGpsKongZhiQiLockCommand:=TRUE;
		END_IF
		IF(BYTE_TO_BOOL(receive_data322[4] AND 2#00000001) )THEN
			VarCanGpsKongZhiQiLockCommand:=FALSE;
		END_IF
	ELSE
		VarCanGpsKongZhiQiLockCommand:=FALSE;
	END_IF

(*开盖锁车*)
	IF(VarCanGpsBEIDONGLockCommand AND  VarCanGpsKaiGaiLockCommand_Enable) AND STATE_WarnKAIGAI THEN
		VarCanGpsKaiGaiLockCommand:=TRUE;
	ELSE
		VarCanGpsKaiGaiLockCommand:=FALSE;
	END_IF
(*天线锁车*)
	IF VarCanGpsBEIDONGLockCommand  AND STATE_WarnTIANXIANoff THEN
		VarCanGpsTianXianLockCommand:=TRUE;
	ELSE
		VarCanGpsTianXianLockCommand:=FALSE;
	END_IF
(*总线故障锁车*)
	IF VarCanGpsBEIDONGLockCommand  AND VarCanGpsTongXunLockCommand_2 THEN
		VarCanGpsTongXunLockCommand:=TRUE;
	ELSE
		VarCanGpsTongXunLockCommand:=FALSE;
	END_IF
(*拔卡故障锁车*)
	IF (VarCanGpsBEIDONGLockCommand AND VarCanGpsBakaLockCommand_Enable)  AND STATE_WarnBAKA THEN
		VarcanGPSbakaCommand:=TRUE;
	ELSE
		VarcanGPSbakaCommand:=FALSE;
	END_IF
(*20天无信号锁车*) 
TIME_60s_3(IN:=NOT TIME_60s_3.Q,PT:=T#60S);
IF NOT STATE_Promoteconnect THEN
	IF TIME_60s_3.Q THEN
		Varjilu_PAR_WorkTime:=Varjilu_PAR_WorkTime+1;
	END_IF
	IF Varjilu_PAR_WorkTime>(TO_UDINT(VarCanGpsYanShiLockCommand_time*30)-1800) THEN  //3天无网络报警
		VarCanNewGpsNoSignalLock_Warning2:=TRUE;
	END_IF
	IF Varjilu_PAR_WorkTime>=(VarCanGpsYanShiLockCommand_time*30) THEN
		STATE_Promoteconnect_20day_2:=TRUE;
		VarCanNewGpsNoSignalLock_Warning2:=FALSE;
	END_IF
ELSE
	Varjilu_PAR_WorkTime:=0;
	STATE_Promoteconnect_20day_2:=FALSE;
	VarCanNewGpsNoSignalLock_Warning2:=FALSE;
END_IF

IF NOT STATE_Promoteconnect THEN
		IF GPS_Time_bool THEN
			IF NOT STATE_Promoteconnect AND Time_bool_once2 AND TIME_5s.Q  THEN
				GPS_Time_Year_Last2 := GPS_Time_Year;
				GPS_Time_Month_Last2 := GPS_Time_Month;
				GPS_Time_Day_Last2  :=  GPS_Time_Day;
				GPS_Time_Hour_Last2 := GPS_Time_Hour;
				GPS_Time_Minute_Last2 := GPS_Time_Minute;
				GPS_Time_Second_Last2 := GPS_Time_Second;
				Time_bool_once2 := FALSE;
			END_IF	
			Time_Sub_Year2 := USINT_TO_SINT(GPS_Time_Year) - USINT_TO_SINT(GPS_Time_Year_Last2);			
			Time_Sub_Month2 := USINT_TO_SINT(GPS_Time_Month) - USINT_TO_SINT(GPS_Time_Month_Last2);	
			Time_Sub_Day2 := USINT_TO_SINT(GPS_Time_Day) - USINT_TO_SINT(GPS_Time_Day_Last2);		
			Time_Sub_Hour2 := USINT_TO_SINT(GPS_Time_Hour) - USINT_TO_SINT(GPS_Time_Hour_Last2);
			Time_Sub_Minute2:=USINT_TO_SINT(GPS_Time_Minute) - USINT_TO_SINT(GPS_Time_Minute_Last2);	
		IF(Time_Sub_Hour2>0) THEN
			Time_hour_Left2:=Time_Sub_Hour2;
		ELSIF(Time_Sub_Day2>0 ) THEN
			Time_hour_Left2:= (Time_Sub_Day2*24)+Time_Sub_Hour2;
		ELSIF(  Time_Sub_Month2>0)THEN
			Time_hour_Left2:= (Time_Sub_Month2*30*24) +(Time_Sub_Day2*24)+Time_Sub_Hour2;
		ELSIF(Time_Sub_Year2>0)THEN
			Time_hour_Left2:= (Time_Sub_Year2*365*24)+(Time_Sub_Month2*30*24) +(Time_Sub_Day2*24)+Time_Sub_Hour2;
		END_IF
		IF GPS_Time_Year>0 OR GPS_Time_Month>0 OR GPS_Time_Day>0 OR GPS_Time_Hour>0 OR  GPS_Time_Minute>0 OR GPS_Time_Second>0  THEN
			IF(TRUE) THEN
				Time_Minute_Left2 :=UINT_TO_INT(VarCanGpsYanShiLockCommand_time)*60 - (Time_hour_Left2 * 60 +Time_Sub_Minute2);
			END_IF		
			IF (Time_Minute_Left2<=4320) THEN   (*3天无信号报警*)	
				VarCanNewGpsNoSignalLock_Warning := TRUE;
			END_IF
			
			IF(Time_Minute_Left2 <= 0) THEN
				STATE_Promoteconnect_20day := TRUE;
				VarCanNewGpsNoSignalLock_Warning := FALSE;
			END_IF
		END_IF
	END_IF
ELSE
	Time_bool_once2:=TRUE;	
	STATE_Promoteconnect_20day:=FALSE;
	VarCanNewGpsNoSignalLock_Warning:=FALSE;
END_IF


IF (VarCanGpsBEIDONGLockCommand AND VarCanGpsYanShiLockCommand_Enable)  AND (STATE_Promoteconnect_20day OR STATE_Promoteconnect_20day_2) THEN
	VarCanGpsYanShiLockCommand:=TRUE;
ELSE
	VarCanGpsYanShiLockCommand:=FALSE;
END_IF
(*B锁车*)
(*		IF(BYTE_TO_BOOL(receive_data322[3] AND 2#00000010) AND NOT BYTE_TO_BOOL(receive_data322[4] AND 2#00000010))THEN
			VarCanGpsLockCommand_B:=TRUE;
		ELSE
			VarCanGpsLockCommand_B:=FALSE;
		END_IF
		IF(BYTE_TO_BOOL(receive_data322[3] AND 2#00000010) )THEN
			VarCanGpsLockCommand_B1:=TRUE;
		ELSE
			VarCanGpsLockCommand_B1:=FALSE;
		END_IF
(*C锁车*)
		IF(BYTE_TO_BOOL(receive_data322[3] AND 2#00000100) AND NOT BYTE_TO_BOOL(receive_data322[4] AND 2#00000100))THEN
			VarCanGpsLockCommand_C:=TRUE;
		ELSE
			VarCanGpsLockCommand_C:=FALSE;
		END_IF
		IF(BYTE_TO_BOOL(receive_data322[3] AND 2#00000100) )THEN
			VarCanGpsLockCommand_C1:=TRUE;
		ELSE
			VarCanGpsLockCommand_C1:=FALSE;
		END_IF
(*D锁车*)
		IF(BYTE_TO_BOOL(receive_data322[3] AND 2#00001000) AND NOT BYTE_TO_BOOL(receive_data322[4] AND 2#00001000))THEN
			VarCanGpsLockCommand_D:=TRUE;
		ELSE
			VarCanGpsLockCommand_D:=FALSE;
		END_IF
		IF(BYTE_TO_BOOL(receive_data322[3] AND 2#00001000) )THEN
			VarCanGpsLockCommand_D1:=TRUE;
		ELSE
			VarCanGpsLockCommand_D1:=FALSE;
		END_IF
(*E锁车*)
		IF(BYTE_TO_BOOL(receive_data322[3] AND 2#00010000) AND NOT BYTE_TO_BOOL(receive_data322[4] AND 2#00010000))THEN
			VarCanGpsLockCommand_E:=TRUE;
		ELSE
			VarCanGpsLockCommand_E:=FALSE;
		END_IF
		IF(BYTE_TO_BOOL(receive_data322[3] AND 2#00010000) )THEN
			VarCanGpsLockCommand_E1:=TRUE;
		ELSE
			VarCanGpsLockCommand_E1:=FALSE;
		END_IF*)
(*BIT0,锁车总使能*)
		IF(BYTE_TO_BOOL(receive_data321[3] AND 2#00000001))THEN
			VarCanGpsenableALLLockCommand:=TRUE;
		END_IF
		IF(BYTE_TO_BOOL(receive_data321[4] AND 2#00000001))THEN
			VarCanGpsenableALLLockCommand:=FALSE;
		END_IF
(*BIT1,被动锁车使能*)
		IF(BYTE_TO_BOOL(receive_data321[3] AND 2#00000010))THEN
			VarCanGpsBEIDONGLockCommand:=TRUE;
		END_IF
		IF(BYTE_TO_BOOL(receive_data321[4] AND 2#00000010))THEN
			VarCanGpsBEIDONGLockCommand:=FALSE;
		END_IF
	
(*BIT2,盲区锁车使能*)
		IF(BYTE_TO_BOOL(receive_data321[3] AND 2#00000100))THEN
			VarCanGpsYanShiLockCommand_Enable:=TRUE;
		END_IF
		IF(BYTE_TO_BOOL(receive_data321[4] AND 2#00000100))THEN
			VarCanGpsYanShiLockCommand_Enable:=FALSE;
		END_IF	
(*BIT3,拆盖锁车使能*)
		IF(BYTE_TO_BOOL(receive_data321[3] AND 2#00001000))THEN
			VarCanGpsKaiGaiLockCommand_Enable:=TRUE;
		END_IF
		IF(BYTE_TO_BOOL(receive_data321[4] AND 2#00001000))THEN
			VarCanGpsKaiGaiLockCommand_Enable:=FALSE;
		END_IF
(*BIT5,拔卡锁车使能*)
		IF(BYTE_TO_BOOL(receive_data321[3] AND 2#00100000))THEN
			VarCanGpsBakaLockCommand_Enable:=TRUE;
		END_IF
		IF(BYTE_TO_BOOL(receive_data321[4] AND 2#00100000))THEN
			VarCanGpsBakaLockCommand_Enable:=FALSE;
		END_IF
(***GPS 锁车***)
(***拆除GPS****)
IF(CAN2_RECE_GPS300.uiAvailable=0) THEN
	GPS_CAN_ERROR_1:=TRUE;
ELSE
	GPS_CAN_ERROR_1:=FALSE;
END_IF

(*10S无数据，总线锁车*)
TIME_2s(IN:=NOT TIME_2s.Q,PT:=T#2S);
IF(TIME_2s.Q)THEN
	IF(VarCanGpsTongXunLockErrorTimer2S<1000)   AND GPS_CAN_ERROR_1  THEN (*控制器与GPS通讯中断报警*)
		VarCanGpsTongXunLockErrorTimer2S:=VarCanGpsTongXunLockErrorTimer2S+1;
		IF(VarCanGpsTongXunLockErrorTimer2S>5)THEN     (*5S*)
			VarCanGpsTongXunLockCommand_2:=TRUE;
			VarCanGpsTongXunLockErrorTimer2S:=0;
		END_IF
	END_IF
END_IF
IF NOT GPS_CAN_ERROR_1 THEN
		VarCanGpsTongXunLockCommand_2:=FALSE;
		VarCanGpsTongXunLockErrorTimer2S:=0;
END_IF
(*真伪校验数据*)
send_data2FF[1]:=UINT_TO_USINT(count MOD 256);(**请求序列号**)
send_data2FF[0]:=UINT_TO_USINT(count/256);
send_data2FF[3]:=DINT_TO_USINT(CANO_engine_hour_h MOD 256);(**校验码1**)
send_data2FF[2]:=DINT_TO_USINT(CANO_engine_hour_h/256);(**校验码2**)
send_data2FF[5]:=UINT_TO_USINT(CANO_engine_hour_m MOD 256);(**校验码3**)
send_data2FF[4]:=UINT_TO_USINT(CANO_engine_hour_m /256);(**校验码4**)
send_data2FF[7]:=UINT_TO_USINT(CANO_Hyd_Tem MOD 256);(**校验码5**)
send_data2FF[6]:=UINT_TO_USINT(CANO_Hyd_Tem/256);(**校验码6**)


data_2FF[0]:=send_data2FF[2];(**校验码1**)
data_2FF[1]:=send_data2FF[3];(**校验码2**)
data_2FF[2]:=send_data2FF[4];(**校验码3**)
data_2FF[3]:=send_data2FF[5];(**校验码4**)
data_2FF[4]:=send_data2FF[6];(**校验码5**)
data_2FF[5]:=send_data2FF[7];(**校验码6**)
uLength01:=UINT_TO_BYTE(6);

swGpsPrivate.swTboxVerification(uData:=data_2FF,uLength:=uLength01,result =>Ver_Output);
SendJIAOYAN_DATA:=send_data2FF[0]*256+send_data2FF[1];

IF SendJIAOYAN_DATA=VarCanGpsJIAOYANNUM THEN
	Judge_Xuhao:=TRUE;
ELSE
	Judge_Xuhao:=FALSE;
END_IF

IF VarCanGpsJIAOYANMA=Ver_Output THEN
	Judge_Jiaoyan:=TRUE;
ELSE
	Judge_Jiaoyan:=FALSE;
END_IF

IF Judge_Xuhao AND Judge_Jiaoyan THEN
	VarCanNewGpsRealFakeResult:=TRUE;
ELSE
	VarCanNewGpsRealFakeResult:=FALSE;
END_IF
TIME_1S_1(IN:=NOT TIME_1S_1.Q,PT:=T#1S);
IF VarCanGpsBEIDONGLockCommand THEN
	IF(TIME_1S_1.Q)THEN
		IF(VarCanGpsFakeErrorTimer1S<1000) AND NOT VarCanNewGpsRealFakeResult THEN
			VarCanGpsFakeErrorTimer1S:=VarCanGpsFakeErrorTimer1S+1;
			IF(VarCanGpsFakeErrorTimer1S>10)THEN  (*10S*)
				VarCanGpsFakeLockCommand:=TRUE;
				VarCanGpsFakeErrorTimer1S:=0;
			END_IF
		END_IF
	END_IF
	IF(VarCanNewGpsRealFakeResult)THEN
		VarCanGpsFakeLockCommand:=FALSE;
		VarCanGpsFakeErrorTimer1S:=0;
	END_IF
ELSE
	VarCanGpsFakeLockCommand:=FALSE;
	VarCanGpsFakeErrorTimer1S:=0;
END_IF
(***所有条件的锁GPS****)

IF((VarCanGpsenableALLLockCommand )AND VarGpsGlobalEnable AND  NOT VarGpsTempUnlockDoing ) THEN    (*锁车全局使能并且没有临时解锁*)
	IF(VarCanGpsKongZhiQiLockCommand OR VarCanGpsYanShiLockCommand OR VarCanGpsTianXianLockCommand OR
		VarCanGpsKaiGaiLockCommand OR   VarcanGPSbakaCommand) THEN
			VarGpsSystemLockedState_bool:=TRUE;
	ELSIF(VarCanGpsTongXunLockCommand OR VarCanGpsFakeLockCommand) THEN
			VarGpsSystemLockedState:=TRUE;
	ELSE
			VarGpsSystemLockedState:=FALSE;
			VarGpsSystemLockedState_bool:=FALSE;
	END_IF
ELSE
	VarGpsSystemLockedState:=FALSE;
	VarGpsSystemLockedState_bool:=FALSE;
END_IF

//延时6小时锁车
	IF((NOT VarGpsSystemLockedState) AND VarGpsSystemLockedState_bool) THEN//已下锁车指令 无锁车时运行 
		IF TIME_60s_3.Q THEN
			Varjilu_PAR_WorkTime2:=Varjilu_PAR_WorkTime2+1;
		END_IF
		IF Varjilu_PAR_WorkTime2>360 THEN  
			VarGpsSystemLockedState:=TRUE;
		END_IF
		IF Varjilu_PAR_WorkTime2<360 THEN
			Time_Minute_Left:=360-Varjilu_PAR_WorkTime2;
		ELSE
			Time_Minute_Left:=0;
		END_IF
	ELSE
		Varjilu_PAR_WorkTime2 := 0;
	END_IF
	


(***GPS 解锁***)
(***网络临时解锁计时***)
(*
TIME_60S(IN:=NOT TIME_60S.Q,PT:=T#60S);
IF(TIME_60S.Q)THEN
	IF(VarGpsPasswordTempUnlockTimer60S<2000) AND VarGpsPasswordTempUnlockEnable  THEN
		VarGpsPasswordTempUnlockTimer60S:=VarGpsPasswordTempUnlockTimer60S+1;
		IF(VarGpsPasswordTempUnlockTimer60S>1440) THEN
			VarGpsPasswordTempUnlockEnable:=FALSE;
			VarGpsPasswordTempUnlockTimer60S:=0;
		END_IF
	END_IF
END_IF
IF(VarGpsPasswordTemporaryCode=9996) AND VarGpsPasswordTempUnlockEnable THEN
		VarGpsPasswordTempUnlockEnable:=FALSE;
		VarGpsPasswordTempUnlockTimer60S:=0;
END_IF*)
(***本地临时解锁*****)
(*IF(VarGpsGlobalEnable)THEN
	IF(VarGpsTempUnlockPassword=9996 AND BYTE_TO_BOOL(VarGpsTempUnlockSelect AND 2#11111111))THEN
		VarGpsTempUnlockSelect:=0;
		VarGpsPasswordTempUnlockTimer60S:=0;
	ELSIF(VarGpsTempUnlockPassword=8402 AND BYTE_TO_BOOL(VarGpsTempUnlockEnable AND 2#00000001))THEN
		VarGpsTempUnlockSelect:=VarGpsTempUnlockSelect OR 2#00000001;
        VarGpsTempUnlockEnable:= VarGpsTempUnlockEnable AND  2#11111110;
	ELSIF(VarGpsTempUnlockPassword=6308 AND BYTE_TO_BOOL(VarGpsTempUnlockEnable AND 2#00000010))THEN
		VarGpsTempUnlockSelect:=VarGpsTempUnlockSelect OR 2#00000010;
        VarGpsTempUnlockEnable:= VarGpsTempUnlockEnable AND  2#11111101;
	ELSIF(VarGpsTempUnlockPassword=8815 AND BYTE_TO_BOOL(VarGpsTempUnlockEnable AND 2#00000100))THEN
		VarGpsTempUnlockSelect:=VarGpsTempUnlockSelect OR 2#00000100;
        VarGpsTempUnlockEnable:= VarGpsTempUnlockEnable AND  2#11111011;
	ELSIF(VarGpsTempUnlockPassword=1678 AND BYTE_TO_BOOL(VarGpsTempUnlockEnable AND 2#00001000))THEN
		VarGpsTempUnlockSelect:=VarGpsTempUnlockSelect OR 2#00001000;
        VarGpsTempUnlockEnable:= VarGpsTempUnlockEnable AND  2#11110111;
	ELSIF(VarGpsTempUnlockPassword=9854 AND BYTE_TO_BOOL(VarGpsTempUnlockEnable AND 2#00010000))THEN
		VarGpsTempUnlockSelect:=VarGpsTempUnlockSelect OR 2#00010000;
        VarGpsTempUnlockEnable:= VarGpsTempUnlockEnable AND  2#11101111;
	ELSIF(VarGpsTempUnlockPassword=11345 AND BYTE_TO_BOOL(VarGpsTempUnlockEnable AND 2#00100000))THEN
		VarGpsTempUnlockSelect:=VarGpsTempUnlockSelect OR 2#00100000;
        VarGpsTempUnlockEnable:= VarGpsTempUnlockEnable AND  2#11011111;
	ELSIF(VarGpsTempUnlockPassword=15342 AND BYTE_TO_BOOL(VarGpsTempUnlockEnable AND 2#01000000))THEN
		VarGpsTempUnlockSelect:=VarGpsTempUnlockSelect OR 2#01000000;
        VarGpsTempUnlockEnable:= VarGpsTempUnlockEnable AND  2#10111111;
	ELSIF(VarGpsTempUnlockPassword=26742 AND BYTE_TO_BOOL(VarGpsTempUnlockEnable AND 2#10000000))THEN
		VarGpsTempUnlockSelect:=VarGpsTempUnlockSelect OR 2#10000000;
        VarGpsTempUnlockEnable:= VarGpsTempUnlockEnable AND  2#01111111;
	END_IF
END_IF
IF(BYTE_TO_BOOL(VarGpsTempUnlockSelect AND 2#11111111) AND VarGpsGlobalEnable)THEN
	IF(VarGpsPasswordTempUnlockTimer60S<=1440)THEN
		VarGpsTempUnlockDoing:=TRUE;
	ELSE
		VarGpsTempUnlockDoing:=FALSE;
		VarGpsTempUnlockSelect:=0;
		VarGpsPasswordTempUnlockTimer60S:=0;
	END_IF
ELSE
	VarGpsTempUnlockDoing:=FALSE;
END_IF
TIME_60s_2(IN:=NOT TIME_60s_2.Q,PT:=T#60S);
IF(TIME_60s_2.Q)THEN
	IF(VarGpsPasswordTempUnlockTimer60S<2000) AND VarGpsTempUnlockDoing    THEN
		VarGpsPasswordTempUnlockTimer60S:=VarGpsPasswordTempUnlockTimer60S+1;
	END_IF
END_IF*)

//临时解锁
IF((VarGpsTempUnlockPassword2=TO_DINT(VarGpsPasswordTemporaryCode)) AND VarGpsGlobalEnable)THEN
	IF NOT VarGpsTempUnlockDoing THEN
		VarGpsTempUnlockDoing:=TRUE;
	END_IF
ELSIF(VarGpsPasswordTemporaryCode=9996)THEN
	IF  VarGpsTempUnlockDoing THEN
		VarGpsTempUnlockDoing:=FALSE;
		VarGpsPasswordTempUnlockTimer60S:=0;
	END_IF
END_IF
TIME_60s_2(IN:=NOT TIME_60s_2.Q,PT:=T#60S);
IF(TIME_60s_2.Q)THEN
	IF(VarGpsPasswordTempUnlockTimer60S<2000) AND VarGpsTempUnlockDoing THEN
		VarGpsPasswordTempUnlockTimer60S:=VarGpsPasswordTempUnlockTimer60S+1;
	END_IF
END_IF
IF(VarGpsPasswordTempUnlockTimer60S>1440)THEN
		VarGpsTempUnlockDoing:=FALSE;
		VarGpsTempUnlockSelect:=0;
		VarGpsPasswordTempUnlockTimer60S:=0;
END_IF

(***永久解锁*****)
(*
GPSYONGJIU(
	Engine_Hour:= (CANO_engine_hour_h), 
	Engine_Minute:=CANO_engine_hour_m , 
	Accum_Depth:= UDINT_TO_DINT(CANO_ACCMUDEPTH)/100, 
	Hyhoil_Tem:= CANO_Hyd_Tem, 
	Water_Tem:=CANO_water_tem , 
	PassWard=> VarGpsYongJiuUnlockPassword);*)

IF (PAR_GPS_ForeverUnlockPassword=(VarGpsYongJiuUnlockPassword2))THEN
	IF(VarGpsGlobalEnable)THEN
		VarGpsGlobalEnable:=FALSE;
	END_IF
ELSIF(PAR_GPS_ForeverUnlockPassword=9996)THEN
	IF(NOT VarGpsGlobalEnable)THEN
		VarGpsGlobalEnable:=TRUE;
	END_IF
END_IF

IF TIME_1000ms.Q THEN
	CAN2_SEND_200(xEnable:= TRUE, eChannel:= 1, udiID:= 16#200, xExtended:=FALSE, usiDLC:=8 , aData:=send_data200);
	CAN2_SEND_201(xEnable:= TRUE, eChannel:= 1, udiID:= 16#201, xExtended:=FALSE, usiDLC:=8 , aData:=send_data201);
	CAN2_SEND_202(xEnable:= TRUE, eChannel:= 1, udiID:= 16#202, xExtended:=FALSE, usiDLC:=8 , aData:=send_data202);
	CAN2_SEND_203(xEnable:= TRUE, eChannel:= 1, udiID:= 16#203, xExtended:=FALSE, usiDLC:=8 , aData:=send_data203);
	CAN2_SEND_204(xEnable:= TRUE, eChannel:= 1, udiID:= 16#204, xExtended:=FALSE, usiDLC:=8 , aData:=send_data204);
	CAN2_SEND_205(xEnable:= TRUE, eChannel:= 1, udiID:= 16#205, xExtended:=FALSE, usiDLC:=8 , aData:=send_data205);
	CAN2_SEND_206(xEnable:= TRUE, eChannel:= 1, udiID:= 16#206, xExtended:=FALSE, usiDLC:=8 , aData:=send_data206);
	CAN2_SEND_207(xEnable:= TRUE, eChannel:= 1, udiID:= 16#207, xExtended:=FALSE, usiDLC:=8 , aData:=send_data207);
	CAN2_SEND_20A(xEnable:= TRUE, eChannel:= 1, udiID:= 16#20A, xExtended:=FALSE, usiDLC:=8 , aData:=send_data20A);
	CAN2_SEND_20B(xEnable:= TRUE, eChannel:= 1, udiID:= 16#20B, xExtended:=FALSE, usiDLC:=8 , aData:=send_data20B);
	CAN2_SEND_20C(xEnable:= TRUE, eChannel:= 1, udiID:= 16#20C, xExtended:=FALSE, usiDLC:=8 , aData:=send_data20C);
	CAN2_SEND_20D(xEnable:= TRUE, eChannel:= 1, udiID:= 16#20D, xExtended:=FALSE, usiDLC:=8 , aData:=send_data20D);
	CAN2_SEND_20E(xEnable:= TRUE, eChannel:= 1, udiID:= 16#20E, xExtended:=FALSE, usiDLC:=8 , aData:=send_data20E);
	CAN2_SEND_211(xEnable:= TRUE, eChannel:= 1, udiID:= 16#211, xExtended:=FALSE, usiDLC:=8 , aData:=send_data211);
	CAN2_SEND_212(xEnable:= TRUE, eChannel:= 1, udiID:= 16#212, xExtended:=FALSE, usiDLC:=8 , aData:=send_data212);
	CAN2_SEND_213(xEnable:= TRUE, eChannel:= 1, udiID:= 16#213, xExtended:=FALSE, usiDLC:=8 , aData:=send_data213);
	CAN2_SEND_214(xEnable:= TRUE, eChannel:= 1, udiID:= 16#214, xExtended:=FALSE, usiDLC:=8 , aData:=send_data214);
	CAN2_SEND_215(xEnable:= TRUE, eChannel:= 1, udiID:= 16#215, xExtended:=FALSE, usiDLC:=8 , aData:=send_data215);
	CAN2_SEND_216(xEnable:= TRUE, eChannel:= 1, udiID:= 16#216, xExtended:=FALSE, usiDLC:=8 , aData:=send_data216);
	CAN2_SEND_217(xEnable:= TRUE, eChannel:= 1, udiID:= 16#217, xExtended:=FALSE, usiDLC:=8 , aData:=send_data217);
	CAN2_SEND_218(xEnable:= TRUE, eChannel:= 1, udiID:= 16#218, xExtended:=FALSE, usiDLC:=8 , aData:=send_data218);
	CAN2_SEND_2F0(xEnable:= TRUE, eChannel:= 1, udiID:= 16#2F0, xExtended:=FALSE, usiDLC:=8 , aData:=send_data2F0);
	CAN2_SEND_2FF(xEnable:= TRUE, eChannel:= 1, udiID:= 16#2FF, xExtended:=FALSE, usiDLC:=8 , aData:=send_data2FF);										
END_IF
IF clear_trig.Q THEN
	CAN2_SEND_2C0(xEnable:= TRUE, eChannel:= 1, udiID:= 16#2C0, xExtended:=FALSE, usiDLC:=8 , aData:=send_data2C0);	
END_IF
(*施工数据，当深度有变化时发送*)(*间隔0.2m*)
(*向远程平台发送施工数据*)
IF(CANO_DEPTH MOD 20)=0 AND (CANO_DEPTH>PAR_DEPTH_VALUE2)THEN
	WORK_SEND:=TRUE;
ELSE
	WORK_SEND:=FALSE;
END_IF
send_trig(CLK:=WORK_SEND);
IF(send_trig.Q)THEN
	CAN2_SEND_280(xEnable:= TRUE, eChannel:= 1, udiID:= 16#280, xExtended:=FALSE, usiDLC:=8 , aData:=send_data280);
	CAN2_SEND_281(xEnable:= TRUE, eChannel:= 1, udiID:= 16#281, xExtended:=FALSE, usiDLC:=8 , aData:=send_data281);
	CAN2_SEND_282(xEnable:= TRUE, eChannel:= 1, udiID:= 16#282, xExtended:=FALSE, usiDLC:=8 , aData:=send_data282);
	CAN2_SEND_283(xEnable:= TRUE, eChannel:= 1, udiID:= 16#283, xExtended:=FALSE, usiDLC:=8 , aData:=send_data283);
	CAN2_SEND_284(xEnable:= TRUE, eChannel:= 1, udiID:= 16#284, xExtended:=FALSE, usiDLC:=8 , aData:=send_data284);
	CAN2_SEND_2B0(xEnable:= TRUE, eChannel:= 1, udiID:= 16#2B0, xExtended:=FALSE, usiDLC:=8 , aData:=send_data2B0);
	CAN2_SEND_2B1(xEnable:= TRUE, eChannel:= 1, udiID:= 16#2B1, xExtended:=FALSE, usiDLC:=8 , aData:=send_data2B1);
END_IF

END_PROGRAM

// StandardPLC/Application/CAN/CanRecover
PROGRAM CanRecover
VAR
	canstatus_0: ifmRCAN.CAN_Status;
	Can0Recover: ifmRCAN.CAN_Recover;
	usiRetryCount_0: USINT;
	xExecute_0: BOOL;
	
	canstatus_1: ifmRCAN.CAN_Status;
	Can1Recover: ifmRCAN.CAN_Recover;
	usiRetryCount_1: USINT;
	xExecute_1: BOOL;
	
	canstatus_2: ifmRCAN.CAN_Status;
	Can2Recover: ifmRCAN.CAN_Recover;
	usiRetryCount_2: USINT;
	xExecute_2: BOOL;
	
	canstatus_3: ifmRCAN.CAN_Status;
	Can3Recover: ifmRCAN.CAN_Recover;
	usiRetryCount_3: USINT;
	xExecute_3: BOOL;
	
END_VAR

(* CAN0 ******************************** *)
canstatus_0(
	xEnable:=TRUE , 
	xError=> , 
	eDiagInfo=> , 
	eChannel:=0 , 
	eBaudrate=> , 
	eBusState=> , 
	uiErrorCntRx=> , 
	uiErrorCntTx=> , 
	xWarningRx=> , 
	xWarningTx=> , 
	udiCountRx=> , 
	usiBusLoad=> );
	IF canstatus_0.usiBusLoad=0   THEN
		xExecute_0:=TRUE;
	ELSE
		xExecute_0:=FALSE;
	END_IF
	IF Can0Recover.usiRetryCount=200 THEN
		xExecute_0:=FALSE;
	END_IF
Can0Recover(
	xExecute:=xExecute_0 , 
	xDone=> , 
	xError=> , 
	eDiagInfo=> , 
	eChannel:=0 , 
	usiNumberRetry:=200 , 
	tInhibitTime:=T#10MS , 
	usiRetryCount=>usiRetryCount_0 );
	
(* CAN1 ******************************** *)
canstatus_1(
	xEnable:=TRUE , 
	xError=> , 
	eDiagInfo=> , 
	eChannel:=1 , 
	eBaudrate=> , 
	eBusState=> , 
	uiErrorCntRx=> , 
	uiErrorCntTx=> , 
	xWarningRx=> , 
	xWarningTx=> , 
	udiCountRx=> , 
	usiBusLoad=> );
	IF canstatus_1.usiBusLoad=0   THEN
		xExecute_1:=TRUE;
	ELSE
		xExecute_1:=FALSE;
	END_IF
	IF Can1Recover.usiRetryCount=200 THEN
		xExecute_1:=FALSE;
	END_IF
Can1Recover(
	xExecute:= xExecute_1, 
	xDone=> , 
	xError=> , 
	eDiagInfo=> , 
	eChannel:=1 , 
	usiNumberRetry:=200 , 
	tInhibitTime:=T#10MS , 
	usiRetryCount=>usiRetryCount_1 );
	
(* CAN2 ******************************** *)
canstatus_2(
	xEnable:=TRUE , 
	xError=> , 
	eDiagInfo=> , 
	eChannel:=2 , 
	eBaudrate=> , 
	eBusState=> , 
	uiErrorCntRx=> , 
	uiErrorCntTx=> , 
	xWarningRx=> , 
	xWarningTx=> , 
	udiCountRx=> , 
	usiBusLoad=> );
	IF canstatus_2.usiBusLoad=0   THEN
		xExecute_2:=TRUE;
	ELSE
		xExecute_2:=FALSE;
	END_IF
	IF Can2Recover.usiRetryCount=200 THEN
		xExecute_2:=FALSE;
	END_IF
Can2Recover(
	xExecute:= xExecute_2, 
	xDone=> , 
	xError=> , 
	eDiagInfo=> , 
	eChannel:=2 , 
	usiNumberRetry:=200 , 
	tInhibitTime:=T#10MS , 
	usiRetryCount=>usiRetryCount_2 );
	
	
(* CAN3 ******************************** *)
canstatus_3(
	xEnable:=TRUE , 
	xError=> , 
	eDiagInfo=> , 
	eChannel:=3 , 
	eBaudrate=> , 
	eBusState=> , 
	uiErrorCntRx=> , 
	uiErrorCntTx=> , 
	xWarningRx=> , 
	xWarningTx=> , 
	udiCountRx=> , 
	usiBusLoad=> );
	IF canstatus_3.usiBusLoad=0   THEN
		xExecute_3:=TRUE;
	ELSE
		xExecute_3:=FALSE;
	END_IF
	IF Can3Recover.usiRetryCount=200 THEN
		xExecute_3:=FALSE;
	END_IF
Can3Recover(
	xExecute:= xExecute_3, 
	xDone=> , 
	xError=> , 
	eDiagInfo=> , 
	eChannel:=3 , 
	usiNumberRetry:=200 , 
	tInhibitTime:=T#10MS , 
	usiRetryCount=>usiRetryCount_3 );

END_PROGRAM

// StandardPLC/Application/CAN/CAN2
PROGRAM CAN2
VAR
	CAN2_INTI: ifmRCAN.CAN_Enable;
	CanERROR_TON1:TON;
	CanERROR_TON2:TON;
	CanERROR_TON3:TON;
	CanERROR_TON4:TON;
	CanERROR_BIAOZHI1:BOOL;	
	CanERROR_BIAOZHI2:BOOL;
	CanERROR_BIAOZHI3:BOOL;	
	CanERROR_BIAOZHI4:BOOL;
	CANI_JOY_Jiao_R_zhongjian:UINT;
	CANI_JOY_Jiao_L_zhongjian:UINT;
	receive_data18ff108c_biaozhi:UINT;
	receive_data0cff108d_biaozhi:UINT;
	CAN3RECEIVE_18FF108C:ifmRCAN.CAN_Rx;
	CAN3RECEIVE_0CFF108D:ifmRCAN.CAN_Rx;
	CAN3RECEIVE_L_Handle:ifmRCAN.CAN_Rx;
	CAN3RECEIVE_R_Handle:ifmRCAN.CAN_Rx;
	CAN3RECEIVE_701:ifmRCAN.CAN_Rx;
	receive_data18ff108c:ARRAY [0..7] OF USINT;
	receive_data0cff108d:ARRAY [0..7] OF USINT;
	receive_data_l_handle:ARRAY [0..7] OF USINT;
	receive_data_r_handle:ARRAY [0..7] OF USINT;
	receive_data701:ARRAY [0..7] OF USINT;
	
	CANI_JOYX_L_biaozhi_zhong:USINT;
	CANI_JOYX_L_zhongjian:USINT;
	CANI_JOYX_L_biaozhi_X_Neg:BOOL;
	CANI_JOYX_L_biaozhi_X_Pos:BOOL;	
	CANI_JOYY_L_biaozhi_zhong:USINT;
	CANI_JOYY_L_zhongjian:USINT;
	CANI_JOYY_L_biaozhi_Y_Neg:BOOL;
	CANI_JOYY_L_biaozhi_Y_Pos:BOOL;	
	CANI_JOYX_R_biaozhi_zhong:USINT;
	CANI_JOYX_R_zhongjian:USINT;
	CANI_JOYX_R_biaozhi_X_Neg:BOOL;
	CANI_JOYX_R_biaozhi_X_Pos:BOOL;	
	CANI_JOYY_R_biaozhi_zhong:USINT;
	CANI_JOYY_R_zhongjian:USINT;
	CANI_JOYY_R_biaozhi_Y_Neg:BOOL;
	CANI_JOYY_R_biaozhi_Y_Pos:BOOL;
		(*IO模块*)
		
	 CAN2_SEND_601:ifmRCAN.CAN_Tx;
	 archives: UINT;
	 CAN1_SEND_000:ifmRCAN.CAN_Tx;
	 CAN1_SEND_201:ifmRCAN.CAN_Tx;
	 CAN1_SEND_601:ifmRCAN.CAN_Tx;
	 send_data000:ARRAY [0..7] OF USINT;
	 send_data201:ARRAY [0..7] OF USINT;
	 send_data601:ARRAY [0..7] OF USINT;
	 init_io:BOOL:=TRUE;
  	 TIME_1s:TON;
	 TIME_100ms:TON;
	 TIME_2s:TON;

	CANI_JOYX_L_biaozhi_X_Neg_Last: BOOL;
	CANI_JOYX_R_Target: UINT;
	JianGE11: UINT:=100;
	CANI_JOYX_L_targat: UINT;
	CANI_JOYX_L_rec: UINT;
	CANI_JOYY_L_rec: UINT;
	CANI_JOYY_R_rec: UINT;
	CANI_JOYX_R_rec: UINT;
	count:int;
	IO_Zhuangtai: USINT;
END_VAR


CAN2_INTI(xEnable:=NOT init_1 , eChannel:=ifmRCAN.ifmDevice.CHAN_2, eBaudrate:=ifmRCAN.ifmDevice.CAN_BAUDRATE.KBAUD_250 );	
(*CAN3口 接左右手柄 左右脚踏 *)
(*右脚踏接收数据*)
CAN3RECEIVE_18FF108C(xEnable:=TRUE , eChannel:= 0, xExtended:= TRUE, aData=> receive_data18ff108c, udiID:= 16#18FF108C);//2-0
(*CAN总线故障保护*)
CanERROR_TON1(IN:=CanERROR_BIAOZHI1,PT:=T#2S);
IF CAN3RECEIVE_18FF108C.uiAvailable = 0 THEN
	CanERROR_BIAOZHI1 :=TRUE;
ELSE
	CanERROR_BIAOZHI1 :=FALSE;
END_IF
IF (CanERROR_TON1.Q) THEN
	receive_data18ff108c[0]:=0;
	receive_data18ff108c[1]:=0;
	receive_data18ff108c[2]:=0;
	receive_data18ff108c[3]:=0;
	receive_data18ff108c[4]:=0;
	receive_data18ff108c[5]:=0;
	receive_data18ff108c[6]:=0;
	receive_data18ff108c[7]:=0;
END_IF

receive_data18ff108c_biaozhi:=receive_data18ff108c[0]+receive_data18ff108c[1]+receive_data18ff108c[2]+receive_data18ff108c[3]
								    +receive_data18ff108c[4]+receive_data18ff108c[5]+receive_data18ff108c[6]+receive_data18ff108c[7];
IF receive_data18ff108c_biaozhi > 0 THEN
	CANI_JOY_Jiao_R_zhongjian:=receive_data18ff108c[0]+receive_data18ff108c[1]*256;
	CANI_JOY_Jiao_R:=UDINT_TO_UINT(REAL_TO_UDINT(UINT_TO_REAL(CANI_JOY_Jiao_R_zhongjian)*50/36));
ELSE
	CANI_JOY_Jiao_R:=2500;
END_IF


(*左脚踏接收数据*)
CAN3RECEIVE_0CFF108D(xEnable:=TRUE , eChannel:= 0, xExtended:= TRUE, aData=> receive_data0cff108d, udiID:= 16#18FF108D);
(*CAN总线故障保护*)
CanERROR_TON2(IN:=CanERROR_BIAOZHI2,PT:=T#2S);
IF CAN3RECEIVE_0CFF108D.uiAvailable = 0 THEN
	CanERROR_BIAOZHI2 :=TRUE;
ELSE
	CanERROR_BIAOZHI2 :=FALSE;
END_IF
IF (CanERROR_TON2.Q) THEN
	receive_data0cff108d[0]:=0;
	receive_data0cff108d[1]:=0;
	receive_data0cff108d[2]:=0;
	receive_data0cff108d[3]:=0;
	receive_data0cff108d[4]:=0;
	receive_data0cff108d[5]:=0;
	receive_data0cff108d[6]:=0;
	receive_data0cff108d[7]:=0;
END_IF
receive_data0cff108d_biaozhi:=receive_data0cff108d[0]+receive_data0cff108d[1]+receive_data0cff108d[2]+receive_data0cff108d[3]
								    +receive_data0cff108d[4]+receive_data0cff108d[5]+receive_data0cff108d[6]+receive_data0cff108d[7];
IF receive_data0cff108d_biaozhi>0 THEN
	CANI_JOY_Jiao_L_zhongjian:=receive_data0cff108d[0]+receive_data0cff108d[1]*256;
	CANI_JOY_Jiao_L:=UDINT_TO_UINT(REAL_TO_UDINT(UINT_TO_REAL(CANI_JOY_Jiao_L_zhongjian)*50/36));
ELSE
	CANI_JOY_Jiao_L:=2500;
END_IF




(*IO模块*)
(*CAN3发送*)
TIME_1s(IN:=init_io,PT:=T#1S);
TIME_100ms(IN:=NOT TIME_100ms.Q,PT:=T#100MS);
TIME_2s(IN:=NOT TIME_2s.Q,PT:=T#2S);
IF TIME_1s.Q  THEN
	init_io:=FALSE;
	archives:=1;
END_IF

//第一步：启动从设备
IF 	TIME_100ms.Q AND archives<20 THEN
 (*   CASE  archives OF
1,2,3,4,5,6,7,8,9,10://第一步：启动从设备
send_data000[0]:=16#01;
send_data000[1]:=16#01;
send_data000[2]:=0;
send_data000[3]:=0;
send_data000[4]:=0;
send_data000[5]:=0;
send_data000[6]:=0;
send_data000[7]:=0;
CAN1_SEND_000(xEnable:=TRUE, eChannel:=2 , udiID:= 16#000, xExtended:=FALSE, usiDLC:=2 , aData:=send_data000 );
11,12://第二步：设定数字量输入发送周期
send_data601[0]:=16#2B;
send_data601[1]:=16#00;
send_data601[2]:=16#18;
send_data601[3]:=16#05;
send_data601[4]:=16#EB;
send_data601[5]:=16#03;
send_data601[6]:=16#00;
send_data601[7]:=16#00;
CAN2_SEND_601(xEnable:=TRUE, eChannel:=2 , udiID:= 16#601, xExtended:=FALSE, usiDLC:=8 , aData:=send_data601 );
13,14://设定模拟量输入周期
send_data601[0]:=16#2B;
send_data601[1]:=16#01;
send_data601[2]:=16#18;
send_data601[3]:=16#05;
send_data601[4]:=16#EB;
send_data601[5]:=16#03;
send_data601[6]:=16#00;
send_data601[7]:=16#00;
CAN2_SEND_601(xEnable:=TRUE, eChannel:=2 , udiID:= 16#601, xExtended:=FALSE, usiDLC:=8 , aData:=send_data601 );
15,16,17,18,19,20://第三步：使能输出
send_data601[0]:=16#23;
send_data601[1]:=16#00;
send_data601[2]:=16#14;
send_data601[3]:=16#01;
send_data601[4]:=16#00;
send_data601[5]:=16#00;
send_data601[6]:=16#00;
send_data601[7]:=16#80;
CAN2_SEND_601(xEnable:=TRUE, eChannel:=2 , udiID:= 16#601, xExtended:=FALSE, usiDLC:=8 , aData:=send_data601 );

    END_CASE*)
archives:=archives+1;
END_IF

send_data000[0]:=16#01;
send_data000[1]:=16#00;
send_data000[2]:=0;
send_data000[3]:=0;
send_data000[4]:=0;
send_data000[5]:=0;
send_data000[6]:=0;
send_data000[7]:=0;
CAN1_SEND_000(xEnable:=TIME_2s.Q, eChannel:=2 , udiID:= 16#000, xExtended:=FALSE, usiDLC:=2 , aData:=send_data000 );
send_data601[0]:=16#23;
send_data601[1]:=16#00;
send_data601[2]:=16#14;
send_data601[3]:=16#01;
send_data601[4]:=16#00;
send_data601[5]:=16#00;
send_data601[6]:=16#00;
send_data601[7]:=16#80;
CAN1_SEND_601(xEnable:=TIME_2s.Q, eChannel:=2 , udiID:= 16#601, xExtended:=FALSE, usiDLC:=8 , aData:=send_data601 );

//输入输出———端口1-8,DO1对应端口3开始
IF archives>=20 THEN
send_data201[0]:=PACK(B0:=FALSE,B1:=FALSE,B2:=DOH_Y50,B3:=DOH_Y51,B4:=DOH_Y52,B5:=DOH_Y53,B6:=DOH_Y54,B7:=DOH_Y55);(*输出DO1-DO6*)
send_data201[1]:=PACK(B0:=DOH_Y56,B1:=DOH_Y57,B2:=DOH_Y59,B3:=DOH_JK1,B4:=DOH_JK2,B5:=DOH_JK3,B6:=DOH_JK4,B7:=DOH_70);(*输出DO7-DO14*)
send_data201[2]:=PACK(B0:=DOH_73,B1:=DOH_B1,B2:=0,B3:=0,B4:=0,B5:=0,B6:=0,B7:=0);(*输出DO15-DO22*)
send_data201[3]:=PACK(B0:=0,B1:=0,B2:=0,B3:=FALSE,B4:=FALSE,B5:=FALSE,B6:=FALSE,B7:=FALSE);
send_data201[4]:=16#00;
send_data201[5]:=16#00;
send_data201[6]:=16#00;
send_data201[7]:=16#00;
CAN1_SEND_201(xEnable:=TIME_100ms.Q, eChannel:=2 , udiID:= 16#201, xExtended:=FALSE, usiDLC:=8 , aData:=send_data201 );
END_IF

(*CAN3RECEIVE_701(xEnable:=TRUE , eChannel:= 2, xExtended:= FALSE, aData=> receive_data701, udiID:= 16#701);
IO_Zhuangtai:=SHR(SHL(receive_data701[0],1),1);
//重启节点
IF(IO_Zhuangtai = 4) THEN
	send_data000[0]:=16#81;
	send_data000[1]:=16#01;
	send_data000[2]:=0;
	send_data000[3]:=0;
	send_data000[4]:=0;
	send_data000[5]:=0;
	send_data000[6]:=0;
	send_data000[7]:=0;
	CAN1_SEND_000(xEnable:=TRUE, eChannel:=2 , udiID:= 16#000, xExtended:=FALSE, usiDLC:=2 , aData:=send_data000 );		
END_IF*)

END_PROGRAM

// StandardPLC/Application/CAN/CAN_J
PROGRAM CAN_J
VAR
	CAN2_INTI: ifmRCAN.CAN_Enable;
	CanERROR_TON1:TON;
	CanERROR_TON2:TON;
	CanERROR_TON3:TON;
	CanERROR_TON4:TON;
	CanERROR_BIAOZHI1:BOOL;	
	CanERROR_BIAOZHI2:BOOL;
	CanERROR_BIAOZHI3:BOOL;	
	CanERROR_BIAOZHI4:BOOL;
	CANI_JOY_Jiao_R_zhongjian:UINT;
	CANI_JOY_Jiao_L_zhongjian:UINT;
	receive_data18ff108c_biaozhi:UINT;
	receive_data0cff108d_biaozhi:UINT;
	CAN3RECEIVE_18FF108C:ifmRCAN.CAN_Rx;
	CAN3RECEIVE_0CFF108D:ifmRCAN.CAN_Rx;
	CAN3RECEIVE_L_Handle:ifmRCAN.CAN_Rx;
	CAN3RECEIVE_R_Handle:ifmRCAN.CAN_Rx;
	CAN3RECEIVE_701:ifmRCAN.CAN_Rx;
	receive_data18ff108c:ARRAY [0..7] OF USINT;
	receive_data0cff108d:ARRAY [0..7] OF USINT;
	receive_data_l_handle:ARRAY [0..7] OF USINT;
	receive_data_r_handle:ARRAY [0..7] OF USINT;
	receive_data701:ARRAY [0..7] OF USINT;
	
	CANI_JOYX_L_biaozhi_zhong:BOOL;
	CANI_JOYX_L_zhongjian:UINT;
	CANI_JOYX_L_biaozhi_X_Neg:BOOL;
	CANI_JOYX_L_biaozhi_X_Pos:BOOL;	
	CANI_JOYY_L_biaozhi_zhong:BOOL;
	CANI_JOYY_L_zhongjian:UINT;
	CANI_JOYY_L_biaozhi_Y_Neg:BOOL;
	CANI_JOYY_L_biaozhi_Y_Pos:BOOL;	
	CANI_JOYX_R_biaozhi_zhong:BOOL;
	CANI_JOYX_R_zhongjian:UINT;
	CANI_JOYX_R_biaozhi_X_Neg:BOOL;
	CANI_JOYX_R_biaozhi_X_Pos:BOOL;	
	CANI_JOYY_R_biaozhi_zhong:BOOL;
	CANI_JOYY_R_zhongjian:UINT;
	CANI_JOYY_R_biaozhi_Y_Neg:BOOL;
	CANI_JOYY_R_biaozhi_Y_Pos:BOOL;
	
		(*IO模块*)
		
	 CAN2_SEND_601:ifmRCAN.CAN_Tx;
	 archives: UINT;
	 CAN1_SEND_000:ifmRCAN.CAN_Tx;
	 CAN1_SEND_201:ifmRCAN.CAN_Tx;
	 CAN1_SEND_601:ifmRCAN.CAN_Tx;
	 send_data000:ARRAY [0..7] OF USINT;
	 send_data201:ARRAY [0..7] OF USINT;
	 send_data601:ARRAY [0..7] OF USINT;
	 init_io:BOOL:=TRUE;
  	 TIME_1s:TON;
	 TIME_100ms:TON;
	 TIME_2s:TON;

	CANI_JOYX_L_biaozhi_X_Neg_Last: BOOL;
	CANI_JOYX_R_Target: UINT;
	JianGE11: UINT:=100;
	CANI_JOYX_L_targat: UINT;
	CANI_JOYX_L_rec: UINT;
	CANI_JOYY_L_rec: UINT;
	CANI_JOYY_R_rec: UINT;
	CANI_JOYX_R_rec: UINT;
	count:int;
	IO_Zhuangtai: USINT;
END_VAR

(*左手柄接收数据*)
CAN3RECEIVE_L_Handle(xEnable:=TRUE , eChannel:= 2, xExtended:= TRUE, aData=> receive_data_l_handle, udiID:= 16#0CFDD634);
CanERROR_TON3(IN:=CanERROR_BIAOZHI3,PT:=T#2S);
IF CAN3RECEIVE_L_Handle.uiAvailable = 0 THEN
	CanERROR_BIAOZHI3 :=TRUE;
ELSE
	CanERROR_BIAOZHI3 :=FALSE;
END_IF
IF ( CanERROR_TON3.Q) THEN
	receive_data_l_handle[0]:=0;
	receive_data_l_handle[1]:=0;
	receive_data_l_handle[2]:=0;
	receive_data_l_handle[3]:=0;
	receive_data_l_handle[4]:=0;
	receive_data_l_handle[5]:=0;
	receive_data_l_handle[6]:=0;
	receive_data_l_handle[7]:=0;
END_IF
(*按钮接收*)
	DI_LHandle_SB1:=USINT_TO_BOOL(receive_data_l_handle[5] AND 2#00000100);//左手柄左边上按钮  解锁按键
	DI_LHandle_SB2:=USINT_TO_BOOL(receive_data_l_handle[5] AND 2#00000001);//左手柄左边下按钮  回转解锁
	DI_LHandle_SB3:=USINT_TO_BOOL(receive_data_l_handle[6] AND 2#01000000);//左手柄中间上按键  浮动
	DI_LHandle_SB4:=USINT_TO_BOOL(receive_data_l_handle[6] AND 2#00010000);//左手柄中间下按键  主卷快速
	DI_LHandle_SB5:=USINT_TO_BOOL(receive_data_l_handle[5] AND 2#00010000);//左手柄右边边上按钮
	DI_LHandle_SB6:=USINT_TO_BOOL(receive_data_l_handle[5] AND 2#01000000);//左手柄右边边下按钮
	DI_LHandle_SB7:=USINT_TO_BOOL(receive_data_l_handle[6] AND 2#00000100);//背部按键 自动回转
	(*IF(receive_data_l_handle[3]>20)THEN
		DI_LHandle_SB7:=TRUE;//回转解锁开关
	ELSE
		DI_LHandle_SB7:=FALSE;		
	END_IF*)
	
	DI_LHandle_SB4_UINT:=receive_data_l_handle[3];
(*X轴方向接收*)
CANI_JOYX_L_zhongjian:=SHR(receive_data_l_handle[0],6)+receive_data_l_handle[1]*4;
CANI_JOYX_L_biaozhi_zhong:=USINT_TO_BOOL(receive_data_l_handle[0] AND 2#00000001);(*手柄中位标志*)
CANI_JOYX_L_biaozhi_X_Neg:=USINT_TO_BOOL(receive_data_l_handle[0] AND 2#00000100);(*手柄X-标志*)
CANI_JOYX_L_biaozhi_X_Pos:=USINT_TO_BOOL(receive_data_l_handle[0] AND 2#00010000);(*手柄X+标志*)

	IF CANI_JOYX_L_biaozhi_zhong THEN(*中位标志为1*)
		CANI_JOYX_L:=2500;(*中位时，左手柄X值为2500*)
	ELSIF CANI_JOYX_L_biaozhi_X_Neg THEN(*左X负向向左标志位1*)
		IF CANI_JOYX_L_zhongjian<1000 THEN(*左手柄Y接收的0-1022的值小于1000时*)
			CANI_JOYX_L:=REAL_TO_UINT((1000-CANI_JOYX_L_zhongjian)*25/10);(*左手柄X负向值为1000-（接收的0到1000）*2.5*)
(*X负向，0-1000换算成2500-0，即0对应2500，1000对应0，反过来了一下***)
		ELSE
			CANI_JOYX_L:=0;(*1000-1022时，左手柄X值为最大，0*)
		END_IF
	ELSIF CANI_JOYX_L_biaozhi_X_Pos THEN(*左X正向标志位1*)
		CANI_JOYX_L:=2500+REAL_TO_UINT(CANI_JOYX_L_zhongjian)*25/10;(*左手柄X正向值为1000-（接收的0到1000）*2.5*)
(*X正向，0-1000换算成2500+（0-2500），即0对应2500，1000对应5000*)
	ELSE
		CANI_JOYX_L:=2500;(*如果俩中位，正负向标志位都不为1，则置为中位*)
	END_IF



(*Y轴方向接收*)
CANI_JOYY_L_zhongjian:=SHR(receive_data_l_handle[2],6)+receive_data_l_handle[3]*4;
CANI_JOYY_L_biaozhi_zhong:=USINT_TO_BOOL(receive_data_l_handle[2] AND 2#00000001);(*手柄Y-标志*)
CANI_JOYY_L_biaozhi_Y_Neg:=USINT_TO_BOOL(receive_data_l_handle[2] AND 2#00000100);(*手柄Y-标志*)
CANI_JOYY_L_biaozhi_Y_Pos:=USINT_TO_BOOL(receive_data_l_handle[2] AND 2#00010000);(*手柄Y+标志*)

	IF CANI_JOYY_L_biaozhi_zhong THEN(*中位标志为1*)
		CANI_JOYY_L:=2500;(*中位时，左手柄Y值为2500*)
	ELSIF CANI_JOYY_L_biaozhi_Y_Neg THEN(*左Y负向向左标志位1*)
		IF CANI_JOYY_L_zhongjian<1000 THEN(*左手柄Y接收的0-1022的值小于1000时*)
			CANI_JOYY_L:=REAL_TO_UINT((1000-CANI_JOYY_L_zhongjian)*25/10);(*左手柄Y负向值为1000-（接收的0到1000）*2.5*)
(*Y负向，0-1000换算成2500-0，即0对应2500，1000对应0，反过来了一下***)
		ELSE
			CANI_JOYY_L:=0;(*1000-1022时，左手柄Y值为最大，0*)
		END_IF
	ELSIF CANI_JOYY_L_biaozhi_Y_Pos THEN(*左Y正向标志位1*)
		CANI_JOYY_L:=2500+REAL_TO_UINT(CANI_JOYY_L_zhongjian)*25/10;(*左手柄Y正向值为1000-（接收的0到1000）*2.5*)
(*Y正向，0-1000换算成2500+（0-2500），即0对应2500，1000对应5000*)
	ELSE
		CANI_JOYY_L:=2500;(*如果俩中位，正负向标志位都不为1，则置为中位*)
	END_IF


(*右手柄接收数据*)
CAN3RECEIVE_R_Handle(xEnable:=TRUE , eChannel:= 2, xExtended:= TRUE, aData=> receive_data_r_handle, udiID:= 16#0CFDD633);
(*CAN总线故障保护*)
CanERROR_TON4(IN:=CanERROR_BIAOZHI4,PT:=T#2S);
IF CAN3RECEIVE_R_Handle.uiAvailable = 0 THEN
	CanERROR_BIAOZHI4 :=TRUE;
ELSE
	CanERROR_BIAOZHI4 :=FALSE;
END_IF

IF ( CanERROR_TON4.Q) THEN
	receive_data_r_handle[0]:=0;
	receive_data_r_handle[1]:=0;
	receive_data_r_handle[2]:=0;
	receive_data_r_handle[3]:=0;
	receive_data_r_handle[4]:=0;
	receive_data_r_handle[5]:=0;
	receive_data_r_handle[6]:=0;
	receive_data_r_handle[7]:=0;
END_IF

(*按钮接收*)
DI_RHandle_SB5:=BYTE_TO_BOOL(receive_data_r_handle[5] AND 2#00000100);(*SB5*)//右手柄左上按键 变幅副卷切换
DI_RHandle_SB6:=BYTE_TO_BOOL(receive_data_r_handle[5] AND 2#00000001);(*SB6*)//右手柄左下按键 动力头抛土
DI_RHandle_SB7:=BYTE_TO_BOOL(receive_data_r_handle[6] AND 2#01000000);(*SB7*)//右手柄中上按键 加压快
DI_RHandle_SB8A:=BYTE_TO_BOOL(receive_data_r_handle[6] AND 2#00010000);(*SB8A*)//备用
DI_RHandle_SB8B:=USINT_TO_BOOL(receive_data_r_handle[5] AND 2#00010000);(*SB8B*)
DI_RHandle_SB1:=USINT_TO_BOOL(receive_data_r_handle[5] AND 2#01000000);
DI_RHandle_SB2:=USINT_TO_BOOL(receive_data_r_handle[6] AND 2#00000100);

//加压快 模拟量按钮


	DI_RHandle_SB7_UINT:=receive_data_r_handle[3];


	
(*X轴方向接收*)
CANI_JOYX_R_zhongjian:=SHR(receive_data_r_handle[0],6)+receive_data_r_handle[1]*4;
CANI_JOYX_R_biaozhi_zhong:=BYTE_TO_BOOL(receive_data_r_handle[0] AND 2#00000001);(*手柄中位标志*)
CANI_JOYX_R_biaozhi_X_Neg:=USINT_TO_BOOL(receive_data_r_handle[0] AND 2#00000100);(*手柄X-标志*)
CANI_JOYX_R_biaozhi_X_Pos:=USINT_TO_BOOL(receive_data_r_handle[0] AND 2#00010000);(*手柄X+标志*)
IF CANI_JOYX_R_biaozhi_zhong THEN
		CANI_JOYX_R:=2500;
	ELSIF CANI_JOYX_R_biaozhi_X_Neg THEN
		IF CANI_JOYX_R_zhongjian<1000 THEN
			CANI_JOYX_R:=REAL_TO_UINT((1000-CANI_JOYX_R_zhongjian)*25/10);
		ELSE
			CANI_JOYX_R:=0;
		END_IF
	ELSIF CANI_JOYX_R_biaozhi_X_Pos THEN
		CANI_JOYX_R:=2500+REAL_TO_UINT(CANI_JOYX_R_zhongjian)*25/10;
	ELSE
		CANI_JOYX_R:=2500;
	END_IF
(*Y轴方向接收*)
CANI_JOYY_R_zhongjian:=SHR(receive_data_r_handle[2],6)+receive_data_r_handle[3]*4;
CANI_JOYY_R_biaozhi_zhong:=BYTE_TO_BOOL(receive_data_r_handle[2] AND 2#00000001);(*手柄中位标志*)
CANI_JOYY_R_biaozhi_Y_Neg:=USINT_TO_BOOL(receive_data_r_handle[2] AND 2#00000100);(*手柄Y-标志*)
CANI_JOYY_R_biaozhi_Y_Pos:=USINT_TO_BOOL(receive_data_r_handle[2] AND 2#00010000);(*手柄Y+标志*)

	IF CANI_JOYY_R_biaozhi_zhong THEN
		CANI_JOYY_R:=2500;
	ELSIF CANI_JOYY_R_biaozhi_Y_Neg THEN
		IF CANI_JOYY_R_zhongjian<1000 THEN
			CANI_JOYY_R:=REAL_TO_UINT((1000-CANI_JOYY_R_zhongjian)*25/10);
		ELSE
			CANI_JOYY_R:=0;
		END_IF
	ELSIF CANI_JOYY_R_biaozhi_Y_Pos THEN
		CANI_JOYY_R:=2500+REAL_TO_UINT(CANI_JOYY_R_zhongjian)*25/10;
	ELSE
		CANI_JOYY_R:=2500;
	END_IF

END_PROGRAM

// StandardPLC/Application/MOVE/control
PROGRAM control
VAR
	
	DI_PWM_JOYX_L: BOOL;
	DI_PWM_JOYY_L: BOOL;
	DI_PWM_JOYX_R: BOOL;
	DI_PWM_JOYY_R: BOOL;
	DI_PWM_JOY_Jiao_R: BOOL;
	DI_PWM_JOY_Jiao_L: BOOL;
	Rotation_move: BOOL;
	MainWinch_move:BOOL;
	PowerHead_move:BOOL;
	JiaYa_move: BOOL;
	LvZhang_move: BOOL;
	BianFu_move:BOOL;
	ViceWinch_move: BOOL;
	LeftMove_move:BOOL;
	RightMove_move:BOOL;
	SPEED_CASE:USINT;
	Enginer_Power:UINT;
	
	PWM_Y1_Target: UINT;	
	PWM_Y2_Target: UINT;	
	
	PWM_Y1_Target_MAX: UINT;
	PWM_Y2_Target_MAX: UINT;
	Hydraulic_Power2:UINT;
	Hydraulic_Power1:UINT;
	Hydraulic_Power:UINT;
	Enginer_Rat: UINT;
	MainPump_Pressure_Taget:UINT;
	Coe_valve: REAL;	
	MainPump_Pressure: UINT;
	Pressure_Coe: REAL;
	PWM_Y1_Target_1: UINT;
	Single_move:BOOL;
	PWM_Y1_Target_OutPut: UINT;
	PWM_Y2_Target_OutPut: UINT;
	PWM_Y34_SET_Target: UINT:=0;
	//PWM_Y33_SET_Target: UINT:=1100;
	

	DonglitouBlink:BLINK;
	DonglitouBlink_biaozhi:BOOL;
	DOH_Y50_1: BOOL;
	Rotation_late:TOF;
	MainPump_Pressure_Taget1000:UINT:=220;
	MainPump_Pressure_Taget1200:UINT:=360;
	MainPump_Pressure_Taget1450:UINT:=420;
	MainPump_Pressure_Taget1600:UINT:=420;
	MainPump_Pressure_Taget1750:UINT:=400;
	MainPump_Pressure_Taget1900:UINT:=360;
	Pressure_Coe_Taget: REAL;
	JianGE1: REAL:=1;
	JianGE2: REAL:=0.005;
	JianGE3: REAL:=3;
	TIME_100ms:TON;
	MainPump_Pressure_last: UINT;
	MainPump_Pressure_last1: UINT;
	TIME_LvBo1:TON;
	TIME_LvBo2:TON;
	TIME_LvBo3:TON;
	MainPump_Pressure_Subtract: INT;
	MainPump_Pressure_ChangeBool: BOOL;
	MainPump_Pressure_ChangeBool1:BOOL;
	PWM_Y2_Target_fuhe: UINT;
	PWM_Y1_Target_fuhe: UINT;
	EngineSpeedSub: UINT;
	PWM_Y23_SET_Taget: UINT;
	PWM_Y24_SET_Taget: UINT;
	CANO_DonglitouPressure_last: UINT;
	DonglitouPressureSub:INT;
	DonglitouPressure_ChangeBool: BOOL;
	JieSuoBool: BOOL;
	ECO_Press_Target1000: UINT:=50;
	ECO_Press_Target1200: UINT:=50;
	ECO_Press_Target1400: UINT:=50;
	ECO_Press_Target1600: UINT:=50;
	ECO_Press_Target1800: UINT:=50;
	ECO_Press_Target1900: UINT:=50;
	
	HELIU_Press_Target1000: UINT:=80;
	HELIU_Press_Target1200: UINT:=80;
	HELIU_Press_Target1400: UINT:=80;
	HELIU_Press_Target1600: UINT:=80;
	HELIU_Press_Target1800: UINT:=80;
	HELIU_Press_Target1900: UINT:=80;
	PWM_Y2_Target_P: UINT;
	PWM_JOY_P_W: UINT;
	XISHU1: REAL:=0.6;
	BiaoZHI_MainWinchUp: BOOL;
	JianGE6:REAL:=2;
	PWM_Y5_SET_Target: UINT;
	PWM_Y6_SET_Target: UINT;
	PWM_Y15_SET_Target: UINT;
	PWM_Y16_SET_Target: UINT;
	PWM_Y5_SET_Target1: INT;
	PWM_Y6_SET_Target1: INT;
	PWM_Y15_SET_Target1: INT;
	PWM_Y16_SET_Target1: INT;
	PWM_Y8_SET_Target: UINT;
	PWM_Y10_SET_Target: UINT;
	PWM_Y7_SET_Target: UINT;
	PWM_Y9_SET_Target: UINT;
	PWM_Y8_SET_Target1: INT;
	PWM_Y10_SET_Target1: INT;
	PWM_Y7_SET_Target1: INT;
	PWM_Y9_SET_Target1: INT;
	JianGE7: UINT:=20;
	JianGE8: UINT:=3;
	PWM_Y39_SET_Target: UINT;
	PWM_Y40_SET_Target: UINT;
	ABS_JOY_1: INT;
	PWM_Y61_SET_Tatget: UINT;
	PWM_Y12_SET_Tatget: UINT;
	PWM_Y14_SET_Tatget: UINT;
	PWM_Y60_SET_Tatget: UINT;
	PWM_Y11_SET_Tatget: UINT;
	PWM_Y13_SET_Tatget: UINT;
	PWM_Y61_SET_Tatget1: INT;
	PWM_Y12_SET_Tatget1: INT;
	PWM_Y14_SET_Tatget1: INT;
	PWM_Y60_SET_Tatget1: INT;
	PWM_Y11_SET_Tatget1: INT;
	PWM_Y13_SET_Tatget1: INT;
	JianGE10: UINT:=25;
	yyyy: UINT;
	TIME_200ms:TON;
	TIME_400ms:TON;
	CANI_JOYX_R_last:UINT;
	Sub_Joyx_r: INT;
	Joyx_change_bool: BOOL;
	JianGE12: UINT:=30;
	Sub_Joyx_r_1: INT;
	BIAOzhi1: BOOL;
	R_TRIG_1:R_TRIG;
	R_TRIG_BOOL: BOOL;
	JianGE22: REAL;
	
	
